LIN {X 0,Y 516.696,Z 376.127,A -85,B 0,C 180,E1 -4916.105,E2 -4916.105} C_VEL
LIN {X 0,Y 516.601,Z 376.349,A -85,B 0,C 180,E1 -4917.032,E2 -4917.032} C_VEL
LIN {X 0,Y 516.544,Z 379.132,A -85,B 0,C 180,E1 -4919.774,E2 -4919.774} C_VEL
LIN {X 0,Y 516.549,Z 381.873,A -85,B 0,C 180,E1 -4922.445,E2 -4922.445} C_VEL
LIN {X 0,Y 516.453,Z 384.593,A -85,B 0,C 180,E1 -4925.048,E2 -4925.048} C_VEL
LIN {X 0,Y 516.411,Z 387.453,A -85,B 0,C 180,E1 -4927.735,E2 -4927.735} C_VEL
LIN {X 0,Y 516.331,Z 390.983,A -85,B 0,C 180,E1 -4930.933,E2 -4930.933} C_VEL
LIN {X 0,Y 516.302,Z 393.789,A -85,B 0,C 180,E1 -4933.39,E2 -4933.39} C_VEL
LIN {X 0,Y 516.34,Z 397.21,A -85,B 0,C 180,E1 -4936.207,E2 -4936.207} C_VEL
LIN {X 0,Y 518.472,Z 408.127,A -85,B 0,C 180,E1 -4936.552,E2 -4936.552} C_VEL
LIN {X 0,Y 518.227,Z 421.717,A -85,B 0,C 180,E1 -4937.07,E2 -4937.07} C_VEL
LIN {X 0,Y 518.019,Z 432.766,A -85,B 0,C 180,E1 -4937.643,E2 -4937.643} C_VEL
LIN {X 0,Y 517.71,Z 443.454,A -85,B 0,C 180,E1 -4938.35,E2 -4938.35} C_VEL
LIN {X 0,Y 517.416,Z 454.111,A -85,B 0,C 180,E1 -4939.236,E2 -4939.236} C_VEL
LIN {X 0,Y 517.106,Z 463.696,A -85,B 0,C 180,E1 -4940.219,E2 -4940.219} C_VEL
LIN {X 0,Y 516.91,Z 471.538,A -85,B 0,C 180,E1 -4941.202,E2 -4941.202} C_VEL
LIN {X 0,Y 516.639,Z 479.209,A -85,B 0,C 180,E1 -4942.378,E2 -4942.378} C_VEL
LIN {X 0,Y 516.493,Z 486.233,A -85,B 0,C 180,E1 -4943.751,E2 -4943.751} C_VEL
LIN {X 0,Y 516.319,Z 490.918,A -85,B 0,C 180,E1 -4944.924,E2 -4944.924} C_VEL
LIN {X 0,Y 516.373,Z 494.495,A -85,B 0,C 180,E1 -4946.098,E2 -4946.098} C_VEL
LIN {X 0,Y 516.313,Z 496.349,A -85,B 0,C 180,E1 -4946.879,E2 -4946.879} C_VEL
LIN {X 0,Y 516.261,Z 497.749,A -85,B 0,C 180,E1 -4947.659,E2 -4947.659} C_VEL
LIN {X 0,Y 516.164,Z 499.358,A -85,B 0,C 180,E1 -4949.22,E2 -4949.22} C_VEL
LIN {X 0,Y 516.161,Z 499.594,A -85,B 0,C 180,E1 -4950,E2 -4950} C_VEL
LIN {X 0,Y 516.164,Z 499.412,A -85,B 0,C 180,E1 -4950.78,E2 -4950.78} C_VEL
LIN {X 0,Y 516.262,Z 497.873,A -85,B 0,C 180,E1 -4952.341,E2 -4952.341} C_VEL
LIN {X 0,Y 516.313,Z 496.527,A -85,B 0,C 180,E1 -4953.121,E2 -4953.121} C_VEL
LIN {X 0,Y 516.363,Z 493.686,A -85,B 0,C 180,E1 -4954.293,E2 -4954.293} C_VEL
LIN {X 0,Y 516.404,Z 489.833,A -85,B 0,C 180,E1 -4955.467,E2 -4955.467} C_VEL
LIN {X 0,Y 516.498,Z 483.973,A -85,B 0,C 180,E1 -4956.823,E2 -4956.823} C_VEL
LIN {X 0,Y 516.73,Z 477.373,A -85,B 0,C 180,E1 -4958.014,E2 -4958.014} C_VEL
LIN {X 0,Y 516.885,Z 469.272,A -85,B 0,C 180,E1 -4959.193,E2 -4959.193} C_VEL
LIN {X 0,Y 517.196,Z 460.967,A -85,B 0,C 180,E1 -4960.175,E2 -4960.175} C_VEL
LIN {X 0,Y 517.521,Z 450.709,A -85,B 0,C 180,E1 -4961.158,E2 -4961.158} C_VEL
LIN {X 0,Y 517.828,Z 440.101,A -85,B 0,C 180,E1 -4961.976,E2 -4961.976} C_VEL
LIN {X 0,Y 518.061,Z 429.415,A -85,B 0,C 180,E1 -4962.636,E2 -4962.636} C_VEL
LIN {X 0,Y 518.325,Z 416.909,A -85,B 0,C 180,E1 -4963.227,E2 -4963.227} C_VEL
LIN {X 0,Y 518.289,Z 407.077,A -85,B 0,C 180,E1 -4963.578,E2 -4963.578} C_VEL
LIN {X 0,Y 516.314,Z 396.997,A -85,B 0,C 180,E1 -4963.906,E2 -4963.906} C_VEL
LIN {X 0,Y 516.316,Z 393.895,A -85,B 0,C 180,E1 -4966.61,E2 -4966.61} C_VEL
LIN {X 0,Y 516.331,Z 391.104,A -85,B 0,C 180,E1 -4969.067,E2 -4969.067} C_VEL
LIN {X 0,Y 516.358,Z 388.318,A -85,B 0,C 180,E1 -4971.561,E2 -4971.561} C_VEL
LIN {X 0,Y 516.434,Z 385.383,A -85,B 0,C 180,E1 -4974.247,E2 -4974.247} C_VEL
LIN {X 0,Y 516.479,Z 382.856,A -85,B 0,C 180,E1 -4976.683,E2 -4976.683} C_VEL
LIN {X 0,Y 516.537,Z 380.02,A -85,B 0,C 180,E1 -4979.45,E2 -4979.45} C_VEL
LIN {X 0,Y 516.572,Z 377.382,A -85,B 0,C 180,E1 -4982.046,E2 -4982.046} C_VEL
LIN {X 0,Y 516.602,Z 376.437,A -85,B 0,C 180,E1 -4982.968,E2 -4982.968} C_VEL
LIN {X 0,Y 516.803,Z 376.111,A -85,B 0,C 180,E1 -4985.319,E2 -4985.319} C_VEL
LIN {X 0,Y 516.884,Z 376.098,A -85,B 0,C 180,E1 -4987.943,E2 -4987.943} C_VEL
LIN {X 0,Y 516.888,Z 376.1,A -85,B 0,C 180,E1 -4990.742,E2 -4990.742} C_VEL
LIN {X 0,Y 516.888,Z 376.098,A -85,B 0,C 180,E1 -4992.831,E2 -4992.831} C_VEL
LIN {X 0,Y 516.899,Z 376.097,A -85,B 0,C 180,E1 -4995.007,E2 -4995.007} C_VEL
LIN {X 0,Y 516.918,Z 376.095,A -85,B 0,C 180,E1 -4998.399,E2 -4998.399} C_VEL
LIN {X 0,Y 516.887,Z 376.098,A -85,B 0,C 180,E1 -5001.284,E2 -5001.284} C_VEL
LIN {X 0,Y 516.892,Z 376.103,A -85,B 0,C 180,E1 -5004.221,E2 -5004.221} C_VEL
LIN {X 0,Y 516.9,Z 376.097,A -85,B 0,C 180,E1 -5007.053,E2 -5007.053} C_VEL
LIN {X 0,Y 516.897,Z 376.099,A -85,B 0,C 180,E1 -5009.796,E2 -5009.796} C_VEL
LIN {X 0,Y 516.931,Z 376.096,A -85,B 0,C 180,E1 -5012.467,E2 -5012.467} C_VEL
LIN {X 0,Y 516.88,Z 376.098,A -85,B 0,C 180,E1 -5015.07,E2 -5015.07} C_VEL
LIN {X 0,Y 516.874,Z 376.101,A -85,B 0,C 180,E1 -5017.622,E2 -5017.622} C_VEL
LIN {X 0,Y 516.938,Z 376.093,A -85,B 0,C 180,E1 -5020.13,E2 -5020.13} C_VEL
LIN {X 0,Y 516.912,Z 376.097,A -85,B 0,C 180,E1 -5022.595,E2 -5022.595} C_VEL
LIN {X 0,Y 516.948,Z 376.093,A -85,B 0,C 180,E1 -5025.03,E2 -5025.03} C_VEL
LIN {X 0,Y 516.971,Z 376.091,A -85,B 0,C 180,E1 -5028.234,E2 -5028.234} C_VEL
LIN {X 0,Y 516.962,Z 376.091,A -85,B 0,C 180,E1 -5031.399,E2 -5031.399} C_VEL
LIN {X 0,Y 517.015,Z 376.083,A -85,B 0,C 180,E1 -5033.757,E2 -5033.757} C_VEL
LIN {X 0,Y 517.086,Z 376.074,A -85,B 0,C 180,E1 -5037.663,E2 -5037.663} C_VEL
LIN {X 0,Y 517.099,Z 376.071,A -85,B 0,C 180,E1 -5040.779,E2 -5040.779} C_VEL
LIN {X 0,Y 517.016,Z 376.082,A -85,B 0,C 180,E1 -5043.117,E2 -5043.117} C_VEL
LIN {X 0,Y 517.015,Z 376.082,A -85,B 0,C 180,E1 -5046.243,E2 -5046.243} C_VEL
LIN {X 0,Y 516.958,Z 376.09,A -85,B 0,C 180,E1 -5049.389,E2 -5049.389} C_VEL
LIN {X 0,Y 516.99,Z 376.089,A -85,B 0,C 180,E1 -5051.824,E2 -5051.824} C_VEL
LIN {X 0,Y 516.95,Z 376.091,A -85,B 0,C 180,E1 -5055.146,E2 -5055.146} C_VEL
LIN {X 0,Y 516.922,Z 376.093,A -85,B 0,C 180,E1 -5058.222,E2 -5058.222} C_VEL
LIN {X 0,Y 516.918,Z 376.098,A -85,B 0,C 180,E1 -5060.701,E2 -5060.701} C_VEL
LIN {X 0,Y 516.896,Z 376.1,A -85,B 0,C 180,E1 -5064.073,E2 -5064.073} C_VEL
LIN {X 0,Y 516.931,Z 376.092,A -85,B 0,C 180,E1 -5066.658,E2 -5066.658} C_VEL
LIN {X 0,Y 516.916,Z 376.096,A -85,B 0,C 180,E1 -5069.524,E2 -5069.524} C_VEL
LIN {X 0,Y 516.9,Z 376.099,A -85,B 0,C 180,E1 -5072.543,E2 -5072.543} C_VEL
LIN {X 0,Y 516.871,Z 376.101,A -85,B 0,C 180,E1 -5075.33,E2 -5075.33} C_VEL
LIN {X 0,Y 516.885,Z 376.1,A -85,B 0,C 180,E1 -5077.943,E2 -5077.943} C_VEL
LIN {X 0,Y 516.887,Z 376.099,A -85,B 0,C 180,E1 -5080.741,E2 -5080.741} C_VEL
LIN {X 0,Y 516.888,Z 376.103,A -85,B 0,C 180,E1 -5082.831,E2 -5082.831} C_VEL
LIN {X 0,Y 516.927,Z 376.095,A -85,B 0,C 180,E1 -5085.01,E2 -5085.01} C_VEL
LIN {X 0,Y 516.92,Z 376.097,A -85,B 0,C 180,E1 -5088.398,E2 -5088.398} C_VEL
LIN {X 0,Y 516.92,Z 376.225,A -85,B 0,C 180,E1 -5091.437,E2 -5091.437} C_VEL
LIN {X 0,Y 518.012,Z 382.521,A -85,B 0,C 180,E1 -5093.83,E2 -5093.83} C_VEL
LIN {X 0,Y 518.066,Z 388.18,A -85,B 0,C 180,E1 -5095.845,E2 -5095.845} C_VEL
LIN {X 0,Y 517.809,Z 396.871,A -85,B 0,C 180,E1 -5098.768,E2 -5098.768} C_VEL
LIN {X 0,Y 517.58,Z 406.618,A -85,B 0,C 180,E1 -5101.959,E2 -5101.959} C_VEL
LIN {X 0,Y 517.332,Z 414.957,A -85,B 0,C 180,E1 -5104.663,E2 -5104.663} C_VEL
LIN {X 0,Y 517.117,Z 424.224,A -85,B 0,C 180,E1 -5107.633,E2 -5107.633} C_VEL
LIN {X 0,Y 516.907,Z 433.491,A -85,B 0,C 180,E1 -5110.542,E2 -5110.542} C_VEL
LIN {X 0,Y 516.714,Z 442.759,A -85,B 0,C 180,E1 -5113.403,E2 -5113.403} C_VEL
LIN {X 0,Y 516.609,Z 451.72,A -85,B 0,C 180,E1 -5116.095,E2 -5116.095} C_VEL
LIN {X 0,Y 518.494,Z 463.261,A -85,B 0,C 180,E1 -5116.403,E2 -5116.403} C_VEL
LIN {X 0,Y 518.294,Z 475.766,A -85,B 0,C 180,E1 -5116.822,E2 -5116.822} C_VEL
LIN {X 0,Y 518.024,Z 487.407,A -85,B 0,C 180,E1 -5117.363,E2 -5117.363} C_VEL
LIN {X 0,Y 517.721,Z 499.455,A -85,B 0,C 180,E1 -5118.102,E2 -5118.102} C_VEL
LIN {X 0,Y 517.44,Z 510.26,A -85,B 0,C 180,E1 -5118.939,E2 -5118.939} C_VEL
LIN {X 0,Y 517.083,Z 519.537,A -85,B 0,C 180,E1 -5119.823,E2 -5119.823} C_VEL
LIN {X 0,Y 516.868,Z 527.99,A -85,B 0,C 180,E1 -5120.806,E2 -5120.806} C_VEL
LIN {X 0,Y 516.641,Z 536.236,A -85,B 0,C 180,E1 -5121.985,E2 -5121.985} C_VEL
LIN {X 0,Y 516.48,Z 543.077,A -85,B 0,C 180,E1 -5123.201,E2 -5123.201} C_VEL
LIN {X 0,Y 516.405,Z 548.949,A -85,B 0,C 180,E1 -5124.533,E2 -5124.533} C_VEL
LIN {X 0,Y 516.343,Z 552.895,A -85,B 0,C 180,E1 -5125.707,E2 -5125.707} C_VEL
LIN {X 0,Y 516.282,Z 555.807,A -85,B 0,C 180,E1 -5126.879,E2 -5126.879} C_VEL
LIN {X 0,Y 516.261,Z 557.196,A -85,B 0,C 180,E1 -5127.659,E2 -5127.659} C_VEL
LIN {X 0,Y 516.16,Z 558.785,A -85,B 0,C 180,E1 -5129.22,E2 -5129.22} C_VEL
LIN {X 0,Y 516.154,Z 559,A -85,B 0,C 180,E1 -5130,E2 -5130} C_VEL
LIN {X 0,Y 516.192,Z 558.185,A -85,B 0,C 180,E1 -5131.56,E2 -5131.56} C_VEL
LIN {X 0,Y 516.261,Z 557.198,A -85,B 0,C 180,E1 -5132.341,E2 -5132.341} C_VEL
LIN {X 0,Y 516.282,Z 555.81,A -85,B 0,C 180,E1 -5133.121,E2 -5133.121} C_VEL
LIN {X 0,Y 516.343,Z 552.896,A -85,B 0,C 180,E1 -5134.293,E2 -5134.293} C_VEL
LIN {X 0,Y 516.405,Z 548.949,A -85,B 0,C 180,E1 -5135.467,E2 -5135.467} C_VEL
LIN {X 0,Y 516.486,Z 543.034,A -85,B 0,C 180,E1 -5136.807,E2 -5136.807} C_VEL
LIN {X 0,Y 516.641,Z 536.237,A -85,B 0,C 180,E1 -5138.015,E2 -5138.015} C_VEL
LIN {X 0,Y 516.868,Z 527.991,A -85,B 0,C 180,E1 -5139.193,E2 -5139.193} C_VEL
LIN {X 0,Y 517.083,Z 519.539,A -85,B 0,C 180,E1 -5140.177,E2 -5140.177} C_VEL
LIN {X 0,Y 517.477,Z 509.096,A -85,B 0,C 180,E1 -5141.159,E2 -5141.159} C_VEL
LIN {X 0,Y 517.73,Z 497.546,A -85,B 0,C 180,E1 -5142.032,E2 -5142.032} C_VEL
LIN {X 0,Y 518.08,Z 485.488,A -85,B 0,C 180,E1 -5142.735,E2 -5142.735} C_VEL
LIN {X 0,Y 518.362,Z 473.168,A -85,B 0,C 180,E1 -5143.276,E2 -5143.276} C_VEL
LIN {X 0,Y 518.314,Z 461.889,A -85,B 0,C 180,E1 -5143.639,E2 -5143.639} C_VEL
LIN {X 0,Y 516.593,Z 451.53,A -85,B 0,C 180,E1 -5143.924,E2 -5143.924} C_VEL
LIN {X 0,Y 516.714,Z 442.759,A -85,B 0,C 180,E1 -5146.596,E2 -5146.596} C_VEL
LIN {X 0,Y 516.906,Z 433.492,A -85,B 0,C 180,E1 -5149.458,E2 -5149.458} C_VEL
LIN {X 0,Y 517.102,Z 423.96,A -85,B 0,C 180,E1 -5152.452,E2 -5152.452} C_VEL
LIN {X 0,Y 517.334,Z 414.957,A -85,B 0,C 180,E1 -5155.336,E2 -5155.336} C_VEL
LIN {X 0,Y 517.607,Z 405.58,A -85,B 0,C 180,E1 -5158.374,E2 -5158.374} C_VEL
LIN {X 0,Y 517.859,Z 395.917,A -85,B 0,C 180,E1 -5161.551,E2 -5161.551} C_VEL
LIN {X 0,Y 518.059,Z 388.196,A -85,B 0,C 180,E1 -5164.154,E2 -5164.154} C_VEL
LIN {X 0,Y 518.018,Z 382.482,A -85,B 0,C 180,E1 -5166.169,E2 -5166.169} C_VEL
LIN {X 0,Y 516.898,Z 376.102,A -85,B 0,C 180,E1 -5168.615,E2 -5168.615} C_VEL
LIN {X 0,Y 516.917,Z 376.1,A -85,B 0,C 180,E1 -5171.775,E2 -5171.775} C_VEL
LIN {X 0,Y 516.926,Z 376.099,A -85,B 0,C 180,E1 -5175.01,E2 -5175.01} C_VEL
LIN {X 0,Y 516.918,Z 376.094,A -85,B 0,C 180,E1 -5178.399,E2 -5178.399} C_VEL
LIN {X 0,Y 516.886,Z 376.098,A -85,B 0,C 180,E1 -5181.284,E2 -5181.284} C_VEL
LIN {X 0,Y 516.89,Z 376.102,A -85,B 0,C 180,E1 -5184.221,E2 -5184.221} C_VEL
LIN {X 0,Y 516.898,Z 376.099,A -85,B 0,C 180,E1 -5187.053,E2 -5187.053} C_VEL
LIN {X 0,Y 516.896,Z 376.096,A -85,B 0,C 180,E1 -5189.796,E2 -5189.796} C_VEL
LIN {X 0,Y 516.932,Z 376.096,A -85,B 0,C 180,E1 -5192.467,E2 -5192.467} C_VEL
LIN {X 0,Y 516.879,Z 376.099,A -85,B 0,C 180,E1 -5195.07,E2 -5195.07} C_VEL
LIN {X 0,Y 516.872,Z 376.103,A -85,B 0,C 180,E1 -5197.622,E2 -5197.622} C_VEL
LIN {X 0,Y 516.936,Z 376.092,A -85,B 0,C 180,E1 -5200.13,E2 -5200.13} C_VEL
LIN {X 0,Y 516.933,Z 376.095,A -85,B 0,C 180,E1 -5202.596,E2 -5202.596} C_VEL
LIN {X 0,Y 516.947,Z 376.09,A -85,B 0,C 180,E1 -5205.03,E2 -5205.03} C_VEL
LIN {X 0,Y 517.009,Z 376.086,A -85,B 0,C 180,E1 -5208.235,E2 -5208.235} C_VEL
LIN {X 0,Y 516.974,Z 376.09,A -85,B 0,C 180,E1 -5211.4,E2 -5211.4} C_VEL
LIN {X 0,Y 517.014,Z 376.082,A -85,B 0,C 180,E1 -5213.757,E2 -5213.757} C_VEL
LIN {X 0,Y 517.088,Z 376.072,A -85,B 0,C 180,E1 -5217.663,E2 -5217.663} C_VEL
LIN {X 0,Y 517.097,Z 376.072,A -85,B 0,C 180,E1 -5220.779,E2 -5220.779} C_VEL
LIN {X 0,Y 517.015,Z 376.085,A -85,B 0,C 180,E1 -5223.117,E2 -5223.117} C_VEL
LIN {X 0,Y 517.014,Z 376.083,A -85,B 0,C 180,E1 -5226.243,E2 -5226.243} C_VEL
LIN {X 0,Y 516.947,Z 376.089,A -85,B 0,C 180,E1 -5229.389,E2 -5229.389} C_VEL
LIN {X 0,Y 516.957,Z 376.092,A -85,B 0,C 180,E1 -5231.807,E2 -5231.807} C_VEL
LIN {X 0,Y 516.949,Z 376.093,A -85,B 0,C 180,E1 -5235.147,E2 -5235.147} C_VEL
LIN {X 0,Y 516.921,Z 376.095,A -85,B 0,C 180,E1 -5238.222,E2 -5238.222} C_VEL
LIN {X 0,Y 516.917,Z 376.096,A -85,B 0,C 180,E1 -5240.701,E2 -5240.701} C_VEL
LIN {X 0,Y 516.895,Z 376.1,A -85,B 0,C 180,E1 -5244.073,E2 -5244.073} C_VEL
LIN {X 0,Y 516.93,Z 376.093,A -85,B 0,C 180,E1 -5246.658,E2 -5246.658} C_VEL
LIN {X 0,Y 516.915,Z 376.096,A -85,B 0,C 180,E1 -5249.524,E2 -5249.524} C_VEL
LIN {X 0,Y 516.899,Z 376.099,A -85,B 0,C 180,E1 -5252.543,E2 -5252.543} C_VEL
LIN {X 0,Y 516.87,Z 376.1,A -85,B 0,C 180,E1 -5255.33,E2 -5255.33} C_VEL
LIN {X 0,Y 516.885,Z 376.1,A -85,B 0,C 180,E1 -5257.943,E2 -5257.943} C_VEL
LIN {X 0,Y 516.888,Z 376.1,A -85,B 0,C 180,E1 -5260.742,E2 -5260.742} C_VEL
LIN {X 0,Y 516.886,Z 376.101,A -85,B 0,C 180,E1 -5262.831,E2 -5262.831} C_VEL
LIN {X 0,Y 516.886,Z 376.102,A -85,B 0,C 180,E1 -5266.097,E2 -5266.097} C_VEL
LIN {X 0,Y 516.919,Z 376.093,A -85,B 0,C 180,E1 -5268.398,E2 -5268.398} C_VEL
LIN {X 0,Y 516.884,Z 376.097,A -85,B 0,C 180,E1 -5270.3,E2 -5270.3} C_VEL
LIN {X 0,Y 516.212,Z 376.184,A -85,B 0,C 180,E1 -5270.95,E2 -5270.95} C_VEL
LIN {X 0,Y 513.358,Z 376.538,A -85,B 0,C 180,E1 -5272.006,E2 -5272.006} C_VEL
LIN {X 0,Y 510.936,Z 376.842,A -85,B 0,C 180,E1 -5272.856,E2 -5272.856} C_VEL
LIN {X 0,Y 509.877,Z 376.973,A -85,B 0,C 180,E1 -5273.512,E2 -5273.512} C_VEL
LIN {X 0,Y 509.781,Z 376.983,A -85,B 0,C 180,E1 -5273.735,E2 -5273.735} C_VEL
LIN {X 0,Y 509.584,Z 377.013,A -85,B 0,C 180,E1 -5276.519,E2 -5276.519} C_VEL
LIN {X 0,Y 509.535,Z 377.482,A -85,B 0,C 180,E1 -5277.457,E2 -5277.457} C_VEL
LIN {X 0,Y 509.477,Z 380.405,A -85,B 0,C 180,E1 -5280.35,E2 -5280.35} C_VEL
LIN {X 0,Y 509.428,Z 383.029,A -85,B 0,C 180,E1 -5282.918,E2 -5282.918} C_VEL
LIN {X 0,Y 509.385,Z 385.793,A -85,B 0,C 180,E1 -5285.59,E2 -5285.59} C_VEL
LIN {X 0,Y 509.309,Z 388.47,A -85,B 0,C 180,E1 -5288.125,E2 -5288.125} C_VEL
LIN {X 0,Y 509.257,Z 391.242,A -85,B 0,C 180,E1 -5290.658,E2 -5290.658} C_VEL
LIN {X 0,Y 509.242,Z 394.076,A -85,B 0,C 180,E1 -5293.153,E2 -5293.153} C_VEL
LIN {X 0,Y 509.28,Z 397.682,A -85,B 0,C 180,E1 -5296.012,E2 -5296.012} C_VEL
LIN {X 0,Y 511.461,Z 408.207,A -85,B 0,C 180,E1 -5296.352,E2 -5296.352} C_VEL
LIN {X 0,Y 511.394,Z 421.035,A -85,B 0,C 180,E1 -5296.843,E2 -5296.843} C_VEL
LIN {X 0,Y 511.133,Z 432.226,A -85,B 0,C 180,E1 -5297.418,E2 -5297.418} C_VEL
LIN {X 0,Y 510.776,Z 443.894,A -85,B 0,C 180,E1 -5298.19,E2 -5298.19} C_VEL
LIN {X 0,Y 510.46,Z 454.549,A -85,B 0,C 180,E1 -5299.088,E2 -5299.088} C_VEL
LIN {X 0,Y 510.137,Z 464.132,A -85,B 0,C 180,E1 -5300.084,E2 -5300.084} C_VEL
LIN {X 0,Y 509.914,Z 471.974,A -85,B 0,C 180,E1 -5301.08,E2 -5301.08} C_VEL
LIN {X 0,Y 509.611,Z 479.644,A -85,B 0,C 180,E1 -5302.273,E2 -5302.273} C_VEL
LIN {X 0,Y 509.445,Z 486.667,A -85,B 0,C 180,E1 -5303.664,E2 -5303.664} C_VEL
LIN {X 0,Y 509.256,Z 491.352,A -85,B 0,C 180,E1 -5304.854,E2 -5304.854} C_VEL
LIN {X 0,Y 509.304,Z 494.928,A -85,B 0,C 180,E1 -5306.044,E2 -5306.044} C_VEL
LIN {X 0,Y 509.259,Z 496.78,A -85,B 0,C 180,E1 -5306.836,E2 -5306.836} C_VEL
LIN {X 0,Y 509.191,Z 498.18,A -85,B 0,C 180,E1 -5307.627,E2 -5307.627} C_VEL
LIN {X 0,Y 509.079,Z 499.79,A -85,B 0,C 180,E1 -5309.209,E2 -5309.209} C_VEL
LIN {X 0,Y 509.075,Z 500.026,A -85,B 0,C 180,E1 -5310,E2 -5310} C_VEL
LIN {X 0,Y 509.078,Z 499.843,A -85,B 0,C 180,E1 -5310.791,E2 -5310.791} C_VEL
LIN {X 0,Y 509.192,Z 498.303,A -85,B 0,C 180,E1 -5312.373,E2 -5312.373} C_VEL
LIN {X 0,Y 509.26,Z 496.956,A -85,B 0,C 180,E1 -5313.165,E2 -5313.165} C_VEL
LIN {X 0,Y 509.291,Z 494.116,A -85,B 0,C 180,E1 -5314.353,E2 -5314.353} C_VEL
LIN {X 0,Y 509.346,Z 490.262,A -85,B 0,C 180,E1 -5315.543,E2 -5315.543} C_VEL
LIN {X 0,Y 509.467,Z 484.594,A -85,B 0,C 180,E1 -5316.879,E2 -5316.879} C_VEL
LIN {X 0,Y 509.702,Z 477.802,A -85,B 0,C 180,E1 -5318.125,E2 -5318.125} C_VEL
LIN {X 0,Y 509.894,Z 469.699,A -85,B 0,C 180,E1 -5319.32,E2 -5319.32} C_VEL
LIN {X 0,Y 510.24,Z 461.391,A -85,B 0,C 180,E1 -5320.315,E2 -5320.315} C_VEL
LIN {X 0,Y 510.578,Z 451.132,A -85,B 0,C 180,E1 -5321.312,E2 -5321.312} C_VEL
LIN {X 0,Y 510.933,Z 439.931,A -85,B 0,C 180,E1 -5322.182,E2 -5322.182} C_VEL
LIN {X 0,Y 511.212,Z 428.023,A -85,B 0,C 180,E1 -5322.909,E2 -5322.909} C_VEL
LIN {X 0,Y 511.496,Z 416.025,A -85,B 0,C 180,E1 -5323.458,E2 -5323.458} C_VEL
LIN {X 0,Y 511.373,Z 407.878,A -85,B 0,C 180,E1 -5323.752,E2 -5323.752} C_VEL
LIN {X 0,Y 509.272,Z 397.377,A -85,B 0,C 180,E1 -5324.103,E2 -5324.103} C_VEL
LIN {X 0,Y 509.308,Z 393.254,A -85,B 0,C 180,E1 -5327.673,E2 -5327.673} C_VEL
LIN {X 0,Y 509.265,Z 389.476,A -85,B 0,C 180,E1 -5331.027,E2 -5331.027} C_VEL
LIN {X 0,Y 509.334,Z 386.717,A -85,B 0,C 180,E1 -5333.588,E2 -5333.588} C_VEL
LIN {X 0,Y 509.412,Z 383.937,A -85,B 0,C 180,E1 -5336.264,E2 -5336.264} C_VEL
LIN {X 0,Y 509.475,Z 381.285,A -85,B 0,C 180,E1 -5338.869,E2 -5338.869} C_VEL
LIN {X 0,Y 509.515,Z 378.508,A -85,B 0,C 180,E1 -5341.612,E2 -5341.612} C_VEL
LIN {X 0,Y 509.538,Z 377.403,A -85,B 0,C 180,E1 -5342.715,E2 -5342.715} C_VEL
LIN {X 0,Y 509.653,Z 377.004,A -85,B 0,C 180,E1 -5344.168,E2 -5344.168} C_VEL
LIN {X 0,Y 509.799,Z 376.985,A -85,B 0,C 180,E1 -5346.91,E2 -5346.91} C_VEL
LIN {X 0,Y 509.838,Z 376.975,A -85,B 0,C 180,E1 -5349.471,E2 -5349.471} C_VEL
LIN {X 0,Y 509.839,Z 376.979,A -85,B 0,C 180,E1 -5352.49,E2 -5352.49} C_VEL
LIN {X 0,Y 509.843,Z 376.978,A -85,B 0,C 180,E1 -5355.33,E2 -5355.33} C_VEL
LIN {X 0,Y 509.86,Z 376.975,A -85,B 0,C 180,E1 -5358.575,E2 -5358.575} C_VEL
LIN {X 0,Y 509.856,Z 376.973,A -85,B 0,C 180,E1 -5361.786,E2 -5361.786} C_VEL
LIN {X 0,Y 509.847,Z 376.975,A -85,B 0,C 180,E1 -5364.623,E2 -5364.623} C_VEL
LIN {X 0,Y 509.866,Z 376.975,A -85,B 0,C 180,E1 -5367.481,E2 -5367.481} C_VEL
LIN {X 0,Y 509.863,Z 376.974,A -85,B 0,C 180,E1 -5370.274,E2 -5370.274} C_VEL
LIN {X 0,Y 509.889,Z 376.972,A -85,B 0,C 180,E1 -5372.944,E2 -5372.944} C_VEL
LIN {X 0,Y 509.856,Z 376.973,A -85,B 0,C 180,E1 -5375.573,E2 -5375.573} C_VEL
LIN {X 0,Y 509.827,Z 376.98,A -85,B 0,C 180,E1 -5378.149,E2 -5378.149} C_VEL
LIN {X 0,Y 509.869,Z 376.973,A -85,B 0,C 180,E1 -5380.682,E2 -5380.682} C_VEL
LIN {X 0,Y 509.879,Z 376.974,A -85,B 0,C 180,E1 -5383.174,E2 -5383.174} C_VEL
LIN {X 0,Y 509.87,Z 376.972,A -85,B 0,C 180,E1 -5385.634,E2 -5385.634} C_VEL
LIN {X 0,Y 509.918,Z 376.965,A -85,B 0,C 180,E1 -5388.875,E2 -5388.875} C_VEL
LIN {X 0,Y 509.927,Z 376.966,A -85,B 0,C 180,E1 -5392.078,E2 -5392.078} C_VEL
LIN {X 0,Y 509.987,Z 376.959,A -85,B 0,C 180,E1 -5394.464,E2 -5394.464} C_VEL
LIN {X 0,Y 510.058,Z 376.949,A -85,B 0,C 180,E1 -5397.631,E2 -5397.631} C_VEL
LIN {X 0,Y 510.069,Z 376.947,A -85,B 0,C 180,E1 -5400.789,E2 -5400.789} C_VEL
LIN {X 0,Y 509.958,Z 376.961,A -85,B 0,C 180,E1 -5403.16,E2 -5403.16} C_VEL
LIN {X 0,Y 509.983,Z 376.958,A -85,B 0,C 180,E1 -5406.33,E2 -5406.33} C_VEL
LIN {X 0,Y 509.921,Z 376.969,A -85,B 0,C 180,E1 -5408.72,E2 -5408.72} C_VEL
LIN {X 0,Y 509.957,Z 376.966,A -85,B 0,C 180,E1 -5411.93,E2 -5411.93} C_VEL
LIN {X 0,Y 509.899,Z 376.97,A -85,B 0,C 180,E1 -5415.242,E2 -5415.242} C_VEL
LIN {X 0,Y 509.867,Z 376.973,A -85,B 0,C 180,E1 -5418.484,E2 -5418.484} C_VEL
LIN {X 0,Y 509.856,Z 376.977,A -85,B 0,C 180,E1 -5421.001,E2 -5421.001} C_VEL
LIN {X 0,Y 509.827,Z 376.979,A -85,B 0,C 180,E1 -5423.564,E2 -5423.564} C_VEL
LIN {X 0,Y 509.917,Z 376.966,A -85,B 0,C 180,E1 -5426.378,E2 -5426.378} C_VEL
LIN {X 0,Y 509.882,Z 376.971,A -85,B 0,C 180,E1 -5428.844,E2 -5428.844} C_VEL
LIN {X 0,Y 509.824,Z 376.978,A -85,B 0,C 180,E1 -5431.59,E2 -5431.59} C_VEL
LIN {X 0,Y 509.852,Z 376.977,A -85,B 0,C 180,E1 -5434.414,E2 -5434.414} C_VEL
LIN {X 0,Y 509.821,Z 376.981,A -85,B 0,C 180,E1 -5437.341,E2 -5437.341} C_VEL
LIN {X 0,Y 509.842,Z 376.975,A -85,B 0,C 180,E1 -5440.382,E2 -5440.382} C_VEL
LIN {X 0,Y 509.828,Z 376.982,A -85,B 0,C 180,E1 -5443.062,E2 -5443.062} C_VEL
LIN {X 0,Y 509.835,Z 376.978,A -85,B 0,C 180,E1 -5445.792,E2 -5445.792} C_VEL
LIN {X 0,Y 509.861,Z 376.975,A -85,B 0,C 180,E1 -5448.575,E2 -5448.575} C_VEL
LIN {X 0,Y 509.855,Z 377.034,A -85,B 0,C 180,E1 -5451.157,E2 -5451.157} C_VEL
LIN {X 0,Y 511.036,Z 383.679,A -85,B 0,C 180,E1 -5453.746,E2 -5453.746} C_VEL
LIN {X 0,Y 511.083,Z 389.074,A -85,B 0,C 180,E1 -5455.681,E2 -5455.681} C_VEL
LIN {X 0,Y 510.85,Z 397.384,A -85,B 0,C 180,E1 -5458.536,E2 -5458.536} C_VEL
LIN {X 0,Y 510.567,Z 407.086,A -85,B 0,C 180,E1 -5461.759,E2 -5461.759} C_VEL
LIN {X 0,Y 510.31,Z 416.281,A -85,B 0,C 180,E1 -5464.727,E2 -5464.727} C_VEL
LIN {X 0,Y 510.081,Z 425.671,A -85,B 0,C 180,E1 -5467.774,E2 -5467.774} C_VEL
LIN {X 0,Y 509.859,Z 434.815,A -85,B 0,C 180,E1 -5470.681,E2 -5470.681} C_VEL
LIN {X 0,Y 509.65,Z 445.407,A -85,B 0,C 180,E1 -5473.99,E2 -5473.99} C_VEL
LIN {X 0,Y 509.563,Z 451.72,A -85,B 0,C 180,E1 -5475.899,E2 -5475.899} C_VEL
LIN {X 0,Y 511.588,Z 464.176,A -85,B 0,C 180,E1 -5476.241,E2 -5476.241} C_VEL
LIN {X 0,Y 511.355,Z 476.979,A -85,B 0,C 180,E1 -5476.69,E2 -5476.69} C_VEL
LIN {X 0,Y 511.034,Z 489.171,A -85,B 0,C 180,E1 -5477.288,E2 -5477.288} C_VEL
LIN {X 0,Y 510.751,Z 499.859,A -85,B 0,C 180,E1 -5477.965,E2 -5477.965} C_VEL
LIN {X 0,Y 510.474,Z 510.261,A -85,B 0,C 180,E1 -5478.786,E2 -5478.786} C_VEL
LIN {X 0,Y 510.072,Z 519.537,A -85,B 0,C 180,E1 -5479.681,E2 -5479.681} C_VEL
LIN {X 0,Y 509.846,Z 527.99,A -85,B 0,C 180,E1 -5480.679,E2 -5480.679} C_VEL
LIN {X 0,Y 509.585,Z 536.235,A -85,B 0,C 180,E1 -5481.873,E2 -5481.873} C_VEL
LIN {X 0,Y 509.419,Z 542.876,A -85,B 0,C 180,E1 -5483.067,E2 -5483.067} C_VEL
LIN {X 0,Y 509.344,Z 548.949,A -85,B 0,C 180,E1 -5484.457,E2 -5484.457} C_VEL
LIN {X 0,Y 509.234,Z 552.894,A -85,B 0,C 180,E1 -5485.647,E2 -5485.647} C_VEL
LIN {X 0,Y 509.2,Z 555.807,A -85,B 0,C 180,E1 -5486.835,E2 -5486.835} C_VEL
LIN {X 0,Y 509.161,Z 557.196,A -85,B 0,C 180,E1 -5487.627,E2 -5487.627} C_VEL
LIN {X 0,Y 509.073,Z 558.786,A -85,B 0,C 180,E1 -5489.209,E2 -5489.209} C_VEL
LIN {X 0,Y 509.065,Z 559,A -85,B 0,C 180,E1 -5490,E2 -5490} C_VEL
LIN {X 0,Y 509.113,Z 558.185,A -85,B 0,C 180,E1 -5491.582,E2 -5491.582} C_VEL
LIN {X 0,Y 509.161,Z 557.198,A -85,B 0,C 180,E1 -5492.373,E2 -5492.373} C_VEL
LIN {X 0,Y 509.2,Z 555.81,A -85,B 0,C 180,E1 -5493.165,E2 -5493.165} C_VEL
LIN {X 0,Y 509.233,Z 552.896,A -85,B 0,C 180,E1 -5494.353,E2 -5494.353} C_VEL
LIN {X 0,Y 509.344,Z 548.949,A -85,B 0,C 180,E1 -5495.543,E2 -5495.543} C_VEL
LIN {X 0,Y 509.41,Z 543.282,A -85,B 0,C 180,E1 -5496.853,E2 -5496.853} C_VEL
LIN {X 0,Y 509.585,Z 536.237,A -85,B 0,C 180,E1 -5498.127,E2 -5498.127} C_VEL
LIN {X 0,Y 509.846,Z 527.991,A -85,B 0,C 180,E1 -5499.321,E2 -5499.321} C_VEL
LIN {X 0,Y 510.071,Z 519.539,A -85,B 0,C 180,E1 -5500.319,E2 -5500.319} C_VEL
LIN {X 0,Y 510.505,Z 509.095,A -85,B 0,C 180,E1 -5501.313,E2 -5501.313} C_VEL
LIN {X 0,Y 510.757,Z 498.326,A -85,B 0,C 180,E1 -5502.143,E2 -5502.143} C_VEL
LIN {X 0,Y 511.08,Z 487.407,A -85,B 0,C 180,E1 -5502.811,E2 -5502.811} C_VEL
LIN {X 0,Y 511.423,Z 475.763,A -85,B 0,C 180,E1 -5503.358,E2 -5503.358} C_VEL
LIN {X 0,Y 511.401,Z 462.803,A -85,B 0,C 180,E1 -5503.802,E2 -5503.802} C_VEL
LIN {X 0,Y 509.552,Z 451.53,A -85,B 0,C 180,E1 -5504.12,E2 -5504.12} C_VEL
LIN {X 0,Y 509.718,Z 441.435,A -85,B 0,C 180,E1 -5507.244,E2 -5507.244} C_VEL
LIN {X 0,Y 509.924,Z 432.168,A -85,B 0,C 180,E1 -5510.155,E2 -5510.155} C_VEL
LIN {X 0,Y 510.125,Z 422.901,A -85,B 0,C 180,E1 -5513.119,E2 -5513.119} C_VEL
LIN {X 0,Y 510.371,Z 413.583,A -85,B 0,C 180,E1 -5516.146,E2 -5516.146} C_VEL
LIN {X 0,Y 510.588,Z 405.374,A -85,B 0,C 180,E1 -5518.8,E2 -5518.8} C_VEL
LIN {X 0,Y 510.861,Z 397.224,A -85,B 0,C 180,E1 -5521.519,E2 -5521.519} C_VEL
LIN {X 0,Y 511.09,Z 388.84,A -85,B 0,C 180,E1 -5524.405,E2 -5524.405} C_VEL
LIN {X 0,Y 511.039,Z 383.669,A -85,B 0,C 180,E1 -5526.253,E2 -5526.253} C_VEL
LIN {X 0,Y 509.86,Z 376.978,A -85,B 0,C 180,E1 -5528.906,E2 -5528.906} C_VEL
LIN {X 0,Y 509.863,Z 376.979,A -85,B 0,C 180,E1 -5531.897,E2 -5531.897} C_VEL
LIN {X 0,Y 509.86,Z 376.981,A -85,B 0,C 180,E1 -5535.332,E2 -5535.332} C_VEL
LIN {X 0,Y 509.86,Z 376.974,A -85,B 0,C 180,E1 -5538.575,E2 -5538.575} C_VEL
LIN {X 0,Y 509.855,Z 376.975,A -85,B 0,C 180,E1 -5541.786,E2 -5541.786} C_VEL
LIN {X 0,Y 509.846,Z 376.976,A -85,B 0,C 180,E1 -5544.623,E2 -5544.623} C_VEL
LIN {X 0,Y 509.864,Z 376.975,A -85,B 0,C 180,E1 -5547.481,E2 -5547.481} C_VEL
LIN {X 0,Y 509.862,Z 376.973,A -85,B 0,C 180,E1 -5550.274,E2 -5550.274} C_VEL
LIN {X 0,Y 509.889,Z 376.971,A -85,B 0,C 180,E1 -5552.945,E2 -5552.945} C_VEL
LIN {X 0,Y 509.855,Z 376.976,A -85,B 0,C 180,E1 -5555.573,E2 -5555.573} C_VEL
LIN {X 0,Y 509.826,Z 376.979,A -85,B 0,C 180,E1 -5558.149,E2 -5558.149} C_VEL
LIN {X 0,Y 509.869,Z 376.974,A -85,B 0,C 180,E1 -5560.682,E2 -5560.682} C_VEL
LIN {X 0,Y 509.888,Z 376.97,A -85,B 0,C 180,E1 -5563.175,E2 -5563.175} C_VEL
LIN {X 0,Y 509.869,Z 376.972,A -85,B 0,C 180,E1 -5565.634,E2 -5565.634} C_VEL
LIN {X 0,Y 509.926,Z 376.965,A -85,B 0,C 180,E1 -5568.875,E2 -5568.875} C_VEL
LIN {X 0,Y 509.956,Z 376.962,A -85,B 0,C 180,E1 -5572.079,E2 -5572.079} C_VEL
LIN {X 0,Y 509.985,Z 376.96,A -85,B 0,C 180,E1 -5574.464,E2 -5574.464} C_VEL
LIN {X 0,Y 510.059,Z 376.947,A -85,B 0,C 180,E1 -5577.631,E2 -5577.631} C_VEL
LIN {X 0,Y 510.068,Z 376.947,A -85,B 0,C 180,E1 -5580.79,E2 -5580.79} C_VEL
LIN {X 0,Y 509.957,Z 376.964,A -85,B 0,C 180,E1 -5583.16,E2 -5583.16} C_VEL
LIN {X 0,Y 509.982,Z 376.96,A -85,B 0,C 180,E1 -5586.33,E2 -5586.33} C_VEL
LIN {X 0,Y 509.913,Z 376.968,A -85,B 0,C 180,E1 -5588.72,E2 -5588.72} C_VEL
LIN {X 0,Y 509.909,Z 376.972,A -85,B 0,C 180,E1 -5591.932,E2 -5591.932} C_VEL
LIN {X 0,Y 509.898,Z 376.971,A -85,B 0,C 180,E1 -5595.242,E2 -5595.242} C_VEL
LIN {X 0,Y 509.871,Z 376.972,A -85,B 0,C 180,E1 -5597.993,E2 -5597.993} C_VEL
LIN {X 0,Y 509.891,Z 376.974,A -85,B 0,C 180,E1 -5600.402,E2 -5600.402} C_VEL
LIN {X 0,Y 509.826,Z 376.978,A -85,B 0,C 180,E1 -5603.564,E2 -5603.564} C_VEL
LIN {X 0,Y 509.916,Z 376.966,A -85,B 0,C 180,E1 -5606.379,E2 -5606.379} C_VEL
LIN {X 0,Y 509.881,Z 376.973,A -85,B 0,C 180,E1 -5608.844,E2 -5608.844} C_VEL
LIN {X 0,Y 509.823,Z 376.978,A -85,B 0,C 180,E1 -5611.59,E2 -5611.59} C_VEL
LIN {X 0,Y 509.851,Z 376.976,A -85,B 0,C 180,E1 -5614.414,E2 -5614.414} C_VEL
LIN {X 0,Y 509.821,Z 376.98,A -85,B 0,C 180,E1 -5617.341,E2 -5617.341} C_VEL
LIN {X 0,Y 509.842,Z 376.976,A -85,B 0,C 180,E1 -5620.382,E2 -5620.382} C_VEL
LIN {X 0,Y 509.826,Z 376.981,A -85,B 0,C 180,E1 -5623.062,E2 -5623.062} C_VEL
LIN {X 0,Y 509.826,Z 376.98,A -85,B 0,C 180,E1 -5625.793,E2 -5625.793} C_VEL
LIN {X 0,Y 509.861,Z 376.972,A -85,B 0,C 180,E1 -5628.575,E2 -5628.575} C_VEL
LIN {X 0,Y 509.854,Z 376.975,A -85,B 0,C 180,E1 -5631.787,E2 -5631.787} C_VEL
LIN {X 0,Y 509.781,Z 376.983,A -85,B 0,C 180,E1 -5633.735,E2 -5633.735} C_VEL
LIN {X 0,Y 509.067,Z 377.098,A -85,B 0,C 180,E1 -5634.395,E2 -5634.395} C_VEL
LIN {X 0,Y 506.12,Z 377.445,A -85,B 0,C 180,E1 -5635.465,E2 -5635.465} C_VEL
LIN {X 0,Y 503.637,Z 377.753,A -85,B 0,C 180,E1 -5636.326,E2 -5636.326} C_VEL
LIN {X 0,Y 502.559,Z 377.91,A -85,B 0,C 180,E1 -5636.991,E2 -5636.991} C_VEL
LIN {X 0,Y 502.465,Z 378.038,A -85,B 0,C 180,E1 -5637.215,E2 -5637.215} C_VEL
LIN {X 0,Y 502.427,Z 380.883,A -85,B 0,C 180,E1 -5640.143,E2 -5640.143} C_VEL
LIN {X 0,Y 502.371,Z 383.283,A -85,B 0,C 180,E1 -5642.506,E2 -5642.506} C_VEL
LIN {X 0,Y 502.299,Z 386.288,A -85,B 0,C 180,E1 -5645.431,E2 -5645.431} C_VEL
LIN {X 0,Y 502.252,Z 388.748,A -85,B 0,C 180,E1 -5647.802,E2 -5647.802} C_VEL
LIN {X 0,Y 502.207,Z 391.512,A -85,B 0,C 180,E1 -5650.375,E2 -5650.375} C_VEL
LIN {X 0,Y 502.187,Z 394.385,A -85,B 0,C 180,E1 -5652.909,E2 -5652.909} C_VEL
LIN {X 0,Y 502.188,Z 397.872,A -85,B 0,C 180,E1 -5655.798,E2 -5655.798} C_VEL
LIN {X 0,Y 504.628,Z 409.413,A -85,B 0,C 180,E1 -5656.189,E2 -5656.189} C_VEL
LIN {X 0,Y 504.469,Z 422.605,A -85,B 0,C 180,E1 -5656.711,E2 -5656.711} C_VEL
LIN {X 0,Y 504.182,Z 434.63,A -85,B 0,C 180,E1 -5657.36,E2 -5657.36} C_VEL
LIN {X 0,Y 503.807,Z 445.615,A -85,B 0,C 180,E1 -5658.126,E2 -5658.126} C_VEL
LIN {X 0,Y 503.475,Z 456.048,A -85,B 0,C 180,E1 -5659.036,E2 -5659.036} C_VEL
LIN {X 0,Y 503.172,Z 464.568,A -85,B 0,C 180,E1 -5659.945,E2 -5659.945} C_VEL
LIN {X 0,Y 502.907,Z 472.41,A -85,B 0,C 180,E1 -5660.955,E2 -5660.955} C_VEL
LIN {X 0,Y 502.599,Z 480.079,A -85,B 0,C 180,E1 -5662.164,E2 -5662.164} C_VEL
LIN {X 0,Y 502.403,Z 487.102,A -85,B 0,C 180,E1 -5663.575,E2 -5663.575} C_VEL
LIN {X 0,Y 502.194,Z 491.786,A -85,B 0,C 180,E1 -5664.781,E2 -5664.781} C_VEL
LIN {X 0,Y 502.237,Z 495.361,A -85,B 0,C 180,E1 -5665.988,E2 -5665.988} C_VEL
LIN {X 0,Y 502.207,Z 497.212,A -85,B 0,C 180,E1 -5666.791,E2 -5666.791} C_VEL
LIN {X 0,Y 502.125,Z 498.612,A -85,B 0,C 180,E1 -5667.594,E2 -5667.594} C_VEL
LIN {X 0,Y 501.995,Z 500.222,A -85,B 0,C 180,E1 -5669.198,E2 -5669.198} C_VEL
LIN {X 0,Y 501.989,Z 500.457,A -85,B 0,C 180,E1 -5670,E2 -5670} C_VEL
LIN {X 0,Y 501.995,Z 500.275,A -85,B 0,C 180,E1 -5670.802,E2 -5670.802} C_VEL
LIN {X 0,Y 502.125,Z 498.733,A -85,B 0,C 180,E1 -5672.407,E2 -5672.407} C_VEL
LIN {X 0,Y 502.207,Z 497.385,A -85,B 0,C 180,E1 -5673.209,E2 -5673.209} C_VEL
LIN {X 0,Y 502.221,Z 494.546,A -85,B 0,C 180,E1 -5674.414,E2 -5674.414} C_VEL
LIN {X 0,Y 502.292,Z 490.692,A -85,B 0,C 180,E1 -5675.621,E2 -5675.621} C_VEL
LIN {X 0,Y 502.395,Z 485.718,A -85,B 0,C 180,E1 -5676.829,E2 -5676.829} C_VEL
LIN {X 0,Y 502.632,Z 479.447,A -85,B 0,C 180,E1 -5678.038,E2 -5678.038} C_VEL
LIN {X 0,Y 502.886,Z 471.595,A -85,B 0,C 180,E1 -5679.249,E2 -5679.249} C_VEL
LIN {X 0,Y 503.273,Z 461.817,A -85,B 0,C 180,E1 -5680.46,E2 -5680.46} C_VEL
LIN {X 0,Y 503.639,Z 451.556,A -85,B 0,C 180,E1 -5681.47,E2 -5681.47} C_VEL
LIN {X 0,Y 503.985,Z 439.842,A -85,B 0,C 180,E1 -5682.39,E2 -5682.39} C_VEL
LIN {X 0,Y 504.327,Z 428.441,A -85,B 0,C 180,E1 -5683.088,E2 -5683.088} C_VEL
LIN {X 0,Y 504.61,Z 416.44,A -85,B 0,C 180,E1 -5683.645,E2 -5683.645} C_VEL
LIN {X 0,Y 504.461,Z 408.671,A -85,B 0,C 180,E1 -5683.931,E2 -5683.931} C_VEL
LIN {X 0,Y 502.195,Z 397.747,A -85,B 0,C 180,E1 -5684.306,E2 -5684.306} C_VEL
LIN {X 0,Y 502.211,Z 393.529,A -85,B 0,C 180,E1 -5687.931,E2 -5687.931} C_VEL
LIN {X 0,Y 502.217,Z 390.666,A -85,B 0,C 180,E1 -5690.478,E2 -5690.478} C_VEL
LIN {X 0,Y 502.244,Z 387.912,A -85,B 0,C 180,E1 -5693.067,E2 -5693.067} C_VEL
LIN {X 0,Y 502.326,Z 385.168,A -85,B 0,C 180,E1 -5695.704,E2 -5695.704} C_VEL
LIN {X 0,Y 502.401,Z 382.44,A -85,B 0,C 180,E1 -5698.4,E2 -5698.4} C_VEL
LIN {X 0,Y 502.478,Z 379.384,A -85,B 0,C 180,E1 -5701.44,E2 -5701.44} C_VEL
LIN {X 0,Y 502.476,Z 377.897,A -85,B 0,C 180,E1 -5703.058,E2 -5703.058} C_VEL
LIN {X 0,Y 502.744,Z 377.861,A -85,B 0,C 180,E1 -5705.954,E2 -5705.954} C_VEL
LIN {X 0,Y 502.805,Z 377.854,A -85,B 0,C 180,E1 -5708.976,E2 -5708.976} C_VEL
LIN {X 0,Y 502.801,Z 377.856,A -85,B 0,C 180,E1 -5712.139,E2 -5712.139} C_VEL
LIN {X 0,Y 502.79,Z 377.856,A -85,B 0,C 180,E1 -5715.47,E2 -5715.47} C_VEL
LIN {X 0,Y 502.824,Z 377.853,A -85,B 0,C 180,E1 -5718.934,E2 -5718.934} C_VEL
LIN {X 0,Y 502.799,Z 377.854,A -85,B 0,C 180,E1 -5722.046,E2 -5722.046} C_VEL
LIN {X 0,Y 502.812,Z 377.85,A -85,B 0,C 180,E1 -5725.035,E2 -5725.035} C_VEL
LIN {X 0,Y 502.788,Z 377.858,A -85,B 0,C 180,E1 -5727.916,E2 -5727.916} C_VEL
LIN {X 0,Y 502.829,Z 377.852,A -85,B 0,C 180,E1 -5730.712,E2 -5730.712} C_VEL
LIN {X 0,Y 502.868,Z 377.845,A -85,B 0,C 180,E1 -5733.439,E2 -5733.439} C_VEL
LIN {X 0,Y 502.781,Z 377.86,A -85,B 0,C 180,E1 -5736.086,E2 -5736.086} C_VEL
LIN {X 0,Y 502.789,Z 377.853,A -85,B 0,C 180,E1 -5738.689,E2 -5738.689} C_VEL
LIN {X 0,Y 502.833,Z 377.851,A -85,B 0,C 180,E1 -5741.248,E2 -5741.248} C_VEL
LIN {X 0,Y 502.854,Z 377.849,A -85,B 0,C 180,E1 -5744.6,E2 -5744.6} C_VEL
LIN {X 0,Y 502.882,Z 377.848,A -85,B 0,C 180,E1 -5748.039,E2 -5748.039} C_VEL
LIN {X 0,Y 502.87,Z 377.844,A -85,B 0,C 180,E1 -5751.157,E2 -5751.157} C_VEL
LIN {X 0,Y 502.933,Z 377.839,A -85,B 0,C 180,E1 -5753.581,E2 -5753.581} C_VEL
LIN {X 0,Y 503.028,Z 377.825,A -85,B 0,C 180,E1 -5757.598,E2 -5757.598} C_VEL
LIN {X 0,Y 503.033,Z 377.829,A -85,B 0,C 180,E1 -5760,E2 -5760} C_VEL
LIN {X 0,Y 503.03,Z 377.823,A -85,B 0,C 180,E1 -5762.402,E2 -5762.402} C_VEL
LIN {X 0,Y 502.933,Z 377.837,A -85,B 0,C 180,E1 -5766.419,E2 -5766.419} C_VEL
LIN {X 0,Y 502.88,Z 377.846,A -85,B 0,C 180,E1 -5768.843,E2 -5768.843} C_VEL
LIN {X 0,Y 502.899,Z 377.843,A -85,B 0,C 180,E1 -5772.1,E2 -5772.1} C_VEL
LIN {X 0,Y 502.854,Z 377.85,A -85,B 0,C 180,E1 -5775.4,E2 -5775.4} C_VEL
LIN {X 0,Y 502.832,Z 377.851,A -85,B 0,C 180,E1 -5778.752,E2 -5778.752} C_VEL
LIN {X 0,Y 502.789,Z 377.855,A -85,B 0,C 180,E1 -5781.311,E2 -5781.311} C_VEL
LIN {X 0,Y 502.781,Z 377.859,A -85,B 0,C 180,E1 -5783.914,E2 -5783.914} C_VEL
LIN {X 0,Y 502.869,Z 377.844,A -85,B 0,C 180,E1 -5786.566,E2 -5786.566} C_VEL
LIN {X 0,Y 502.829,Z 377.853,A -85,B 0,C 180,E1 -5789.288,E2 -5789.288} C_VEL
LIN {X 0,Y 502.788,Z 377.855,A -85,B 0,C 180,E1 -5792.084,E2 -5792.084} C_VEL
LIN {X 0,Y 502.803,Z 377.853,A -85,B 0,C 180,E1 -5794.966,E2 -5794.966} C_VEL
LIN {X 0,Y 502.798,Z 377.855,A -85,B 0,C 180,E1 -5797.954,E2 -5797.954} C_VEL
LIN {X 0,Y 502.823,Z 377.854,A -85,B 0,C 180,E1 -5801.066,E2 -5801.066} C_VEL
LIN {X 0,Y 502.805,Z 377.856,A -85,B 0,C 180,E1 -5804.532,E2 -5804.532} C_VEL
LIN {X 0,Y 502.834,Z 377.853,A -85,B 0,C 180,E1 -5807.864,E2 -5807.864} C_VEL
LIN {X 0,Y 502.82,Z 377.918,A -85,B 0,C 180,E1 -5810.896,E2 -5810.896} C_VEL
LIN {X 0,Y 504.012,Z 384.68,A -85,B 0,C 180,E1 -5813.6,E2 -5813.6} C_VEL
LIN {X 0,Y 504.126,Z 389.447,A -85,B 0,C 180,E1 -5815.338,E2 -5815.338} C_VEL
LIN {X 0,Y 503.876,Z 397.914,A -85,B 0,C 180,E1 -5818.301,E2 -5818.301} C_VEL
LIN {X 0,Y 503.585,Z 406.488,A -85,B 0,C 180,E1 -5821.203,E2 -5821.203} C_VEL
LIN {X 0,Y 503.331,Z 414.728,A -85,B 0,C 180,E1 -5823.906,E2 -5823.906} C_VEL
LIN {X 0,Y 503.141,Z 422.9,A -85,B 0,C 180,E1 -5826.541,E2 -5826.541} C_VEL
LIN {X 0,Y 502.903,Z 432.167,A -85,B 0,C 180,E1 -5829.551,E2 -5829.551} C_VEL
LIN {X 0,Y 502.664,Z 441.435,A -85,B 0,C 180,E1 -5832.506,E2 -5832.506} C_VEL
LIN {X 0,Y 502.506,Z 451.581,A -85,B 0,C 180,E1 -5835.694,E2 -5835.694} C_VEL
LIN {X 0,Y 504.69,Z 465.089,A -85,B 0,C 180,E1 -5836.075,E2 -5836.075} C_VEL
LIN {X 0,Y 504.428,Z 478.108,A -85,B 0,C 180,E1 -5836.555,E2 -5836.555} C_VEL
LIN {X 0,Y 504.055,Z 490.528,A -85,B 0,C 180,E1 -5837.188,E2 -5837.188} C_VEL
LIN {X 0,Y 503.741,Z 501.586,A -85,B 0,C 180,E1 -5837.92,E2 -5837.92} C_VEL
LIN {X 0,Y 503.385,Z 512.467,A -85,B 0,C 180,E1 -5838.83,E2 -5838.83} C_VEL
LIN {X 0,Y 503.024,Z 521.332,A -85,B 0,C 180,E1 -5839.739,E2 -5839.739} C_VEL
LIN {X 0,Y 502.704,Z 530.96,A -85,B 0,C 180,E1 -5840.951,E2 -5840.951} C_VEL
LIN {X 0,Y 502.47,Z 538.621,A -85,B 0,C 180,E1 -5842.162,E2 -5842.162} C_VEL
LIN {X 0,Y 502.275,Z 545.679,A -85,B 0,C 180,E1 -5843.573,E2 -5843.573} C_VEL
LIN {X 0,Y 502.186,Z 550.372,A -85,B 0,C 180,E1 -5844.781,E2 -5844.781} C_VEL
LIN {X 0,Y 502.151,Z 553.958,A -85,B 0,C 180,E1 -5845.987,E2 -5845.987} C_VEL
LIN {X 0,Y 502.121,Z 555.807,A -85,B 0,C 180,E1 -5846.79,E2 -5846.79} C_VEL
LIN {X 0,Y 502.066,Z 557.195,A -85,B 0,C 180,E1 -5847.593,E2 -5847.593} C_VEL
LIN {X 0,Y 501.99,Z 558.786,A -85,B 0,C 180,E1 -5849.198,E2 -5849.198} C_VEL
LIN {X 0,Y 501.98,Z 559,A -85,B 0,C 180,E1 -5850,E2 -5850} C_VEL
LIN {X 0,Y 502.036,Z 558.185,A -85,B 0,C 180,E1 -5851.604,E2 -5851.604} C_VEL
LIN {X 0,Y 502.066,Z 557.198,A -85,B 0,C 180,E1 -5852.407,E2 -5852.407} C_VEL
LIN {X 0,Y 502.121,Z 555.81,A -85,B 0,C 180,E1 -5853.209,E2 -5853.209} C_VEL
LIN {X 0,Y 502.128,Z 552.896,A -85,B 0,C 180,E1 -5854.415,E2 -5854.415} C_VEL
LIN {X 0,Y 502.259,Z 548.949,A -85,B 0,C 180,E1 -5855.621,E2 -5855.621} C_VEL
LIN {X 0,Y 502.336,Z 542.977,A -85,B 0,C 180,E1 -5857.011,E2 -5857.011} C_VEL
LIN {X 0,Y 502.542,Z 536.236,A -85,B 0,C 180,E1 -5858.241,E2 -5858.241} C_VEL
LIN {X 0,Y 502.811,Z 527.991,A -85,B 0,C 180,E1 -5859.453,E2 -5859.453} C_VEL
LIN {X 0,Y 503.065,Z 519.539,A -85,B 0,C 180,E1 -5860.464,E2 -5860.464} C_VEL
LIN {X 0,Y 503.532,Z 509.094,A -85,B 0,C 180,E1 -5861.472,E2 -5861.472} C_VEL
LIN {X 0,Y 503.805,Z 497.501,A -85,B 0,C 180,E1 -5862.372,E2 -5862.372} C_VEL
LIN {X 0,Y 504.216,Z 485.489,A -85,B 0,C 180,E1 -5863.091,E2 -5863.091} C_VEL
LIN {X 0,Y 504.533,Z 473.166,A -85,B 0,C 180,E1 -5863.647,E2 -5863.647} C_VEL
LIN {X 0,Y 504.506,Z 463.717,A -85,B 0,C 180,E1 -5863.969,E2 -5863.969} C_VEL
LIN {X 0,Y 502.505,Z 451.53,A -85,B 0,C 180,E1 -5864.322,E2 -5864.322} C_VEL
LIN {X 0,Y 502.664,Z 441.435,A -85,B 0,C 180,E1 -5867.494,E2 -5867.494} C_VEL
LIN {X 0,Y 502.907,Z 431.827,A -85,B 0,C 180,E1 -5870.559,E2 -5870.559} C_VEL
LIN {X 0,Y 503.189,Z 421.577,A -85,B 0,C 180,E1 -5873.894,E2 -5873.894} C_VEL
LIN {X 0,Y 503.455,Z 411.904,A -85,B 0,C 180,E1 -5877.012,E2 -5877.012} C_VEL
LIN {X 0,Y 503.724,Z 402.43,A -85,B 0,C 180,E1 -5880.151,E2 -5880.151} C_VEL
LIN {X 0,Y 504.033,Z 393.547,A -85,B 0,C 180,E1 -5883.216,E2 -5883.216} C_VEL
LIN {X 0,Y 504.186,Z 386.177,A -85,B 0,C 180,E1 -5885.835,E2 -5885.835} C_VEL
LIN {X 0,Y 503.346,Z 380.852,A -85,B 0,C 180,E1 -5887.905,E2 -5887.905} C_VEL
LIN {X 0,Y 502.808,Z 377.856,A -85,B 0,C 180,E1 -5889.169,E2 -5889.169} C_VEL
LIN {X 0,Y 502.806,Z 377.859,A -85,B 0,C 180,E1 -5892.199,E2 -5892.199} C_VEL
LIN {X 0,Y 502.804,Z 377.861,A -85,B 0,C 180,E1 -5895.468,E2 -5895.468} C_VEL
LIN {X 0,Y 502.823,Z 377.855,A -85,B 0,C 180,E1 -5898.934,E2 -5898.934} C_VEL
LIN {X 0,Y 502.797,Z 377.855,A -85,B 0,C 180,E1 -5902.046,E2 -5902.046} C_VEL
LIN {X 0,Y 502.81,Z 377.853,A -85,B 0,C 180,E1 -5905.035,E2 -5905.035} C_VEL
LIN {X 0,Y 502.786,Z 377.855,A -85,B 0,C 180,E1 -5907.916,E2 -5907.916} C_VEL
LIN {X 0,Y 502.828,Z 377.853,A -85,B 0,C 180,E1 -5910.712,E2 -5910.712} C_VEL
LIN {X 0,Y 502.866,Z 377.844,A -85,B 0,C 180,E1 -5913.439,E2 -5913.439} C_VEL
LIN {X 0,Y 502.78,Z 377.859,A -85,B 0,C 180,E1 -5916.086,E2 -5916.086} C_VEL
LIN {X 0,Y 502.787,Z 377.855,A -85,B 0,C 180,E1 -5918.689,E2 -5918.689} C_VEL
LIN {X 0,Y 502.834,Z 377.85,A -85,B 0,C 180,E1 -5921.248,E2 -5921.248} C_VEL
LIN {X 0,Y 502.826,Z 377.848,A -85,B 0,C 180,E1 -5923.767,E2 -5923.767} C_VEL
LIN {X 0,Y 502.836,Z 377.852,A -85,B 0,C 180,E1 -5926.255,E2 -5926.255} C_VEL
LIN {X 0,Y 502.896,Z 377.841,A -85,B 0,C 180,E1 -5928.717,E2 -5928.717} C_VEL
LIN {X 0,Y 502.906,Z 377.841,A -85,B 0,C 180,E1 -5931.967,E2 -5931.967} C_VEL
LIN {X 0,Y 502.941,Z 377.837,A -85,B 0,C 180,E1 -5934.387,E2 -5934.387} C_VEL
LIN {X 0,Y 503.028,Z 377.823,A -85,B 0,C 180,E1 -5937.598,E2 -5937.598} C_VEL
LIN {X 0,Y 503.031,Z 377.828,A -85,B 0,C 180,E1 -5940,E2 -5940} C_VEL
LIN {X 0,Y 503.026,Z 377.825,A -85,B 0,C 180,E1 -5942.402,E2 -5942.402} C_VEL
LIN {X 0,Y 502.942,Z 377.836,A -85,B 0,C 180,E1 -5945.614,E2 -5945.614} C_VEL
LIN {X 0,Y 502.904,Z 377.841,A -85,B 0,C 180,E1 -5948.033,E2 -5948.033} C_VEL
LIN {X 0,Y 502.881,Z 377.842,A -85,B 0,C 180,E1 -5951.283,E2 -5951.283} C_VEL
LIN {X 0,Y 502.849,Z 377.847,A -85,B 0,C 180,E1 -5954.571,E2 -5954.571} C_VEL
LIN {X 0,Y 502.827,Z 377.85,A -85,B 0,C 180,E1 -5957.908,E2 -5957.908} C_VEL
LIN {X 0,Y 502.833,Z 377.851,A -85,B 0,C 180,E1 -5960.536,E2 -5960.536} C_VEL
LIN {X 0,Y 502.792,Z 377.852,A -85,B 0,C 180,E1 -5963.041,E2 -5963.041} C_VEL
LIN {X 0,Y 502.826,Z 377.854,A -85,B 0,C 180,E1 -5965.677,E2 -5965.677} C_VEL
LIN {X 0,Y 502.844,Z 377.848,A -85,B 0,C 180,E1 -5968.373,E2 -5968.373} C_VEL
LIN {X 0,Y 502.796,Z 377.854,A -85,B 0,C 180,E1 -5971.499,E2 -5971.499} C_VEL
LIN {X 0,Y 502.808,Z 377.856,A -85,B 0,C 180,E1 -5973.994,E2 -5973.994} C_VEL
LIN {X 0,Y 502.781,Z 377.855,A -85,B 0,C 180,E1 -5977.178,E2 -5977.178} C_VEL
LIN {X 0,Y 502.792,Z 377.854,A -85,B 0,C 180,E1 -5980.015,E2 -5980.015} C_VEL
LIN {X 0,Y 502.806,Z 377.854,A -85,B 0,C 180,E1 -5982.199,E2 -5982.199} C_VEL
LIN {X 0,Y 502.789,Z 377.855,A -85,B 0,C 180,E1 -5985.47,E2 -5985.47} C_VEL
LIN {X 0,Y 502.833,Z 377.853,A -85,B 0,C 180,E1 -5987.864,E2 -5987.864} C_VEL
LIN {X 0,Y 502.804,Z 377.853,A -85,B 0,C 180,E1 -5991.024,E2 -5991.024} C_VEL
LIN {X 0,Y 502.742,Z 377.862,A -85,B 0,C 180,E1 -5994.175,E2 -5994.175} C_VEL
LIN {X 0,Y 502.475,Z 377.898,A -85,B 0,C 180,E1 -5997.057,E2 -5997.057} C_VEL
LIN {X 0,Y 502.465,Z 378.038,A -85,B 0,C 180,E1 -5997.215,E2 -5997.215} C_VEL
LIN {X 0,Y 501.775,Z 378.714,A -85,B 0,C 180,E1 -5997.88,E2 -5997.88} C_VEL
LIN {X 0,Y 498.893,Z 380.049,A -85,B 0,C 180,E1 -5998.955,E2 -5998.955} C_VEL
LIN {X 0,Y 496.461,Z 381.154,A -85,B 0,C 180,E1 -5999.821,E2 -5999.821} C_VEL
LIN {X 0,Y 495.411,Z 381.928,A -85,B 0,C 180,E1 -6000.491,E2 -6000.491} C_VEL
LIN {X 0,Y 495.322,Z 382.165,A -85,B 0,C 180,E1 -6000.719,E2 -6000.719} C_VEL
LIN {X 0,Y 495.281,Z 384.855,A -85,B 0,C 180,E1 -6003.376,E2 -6003.376} C_VEL
LIN {X 0,Y 495.223,Z 387.215,A -85,B 0,C 180,E1 -6005.697,E2 -6005.697} C_VEL
LIN {X 0,Y 495.157,Z 389.95,A -85,B 0,C 180,E1 -6008.344,E2 -6008.344} C_VEL
LIN {X 0,Y 495.13,Z 392.759,A -85,B 0,C 180,E1 -6010.945,E2 -6010.945} C_VEL
LIN {X 0,Y 495.09,Z 395.67,A -85,B 0,C 180,E1 -6013.506,E2 -6013.506} C_VEL
LIN {X 0,Y 495.141,Z 398.187,A -85,B 0,C 180,E1 -6015.591,E2 -6015.591} C_VEL
LIN {X 0,Y 497.688,Z 410.246,A -85,B 0,C 180,E1 -6016.006,E2 -6016.006} C_VEL
LIN {X 0,Y 497.597,Z 423.05,A -85,B 0,C 180,E1 -6016.524,E2 -6016.524} C_VEL
LIN {X 0,Y 497.303,Z 434.502,A -85,B 0,C 180,E1 -6017.145,E2 -6017.145} C_VEL
LIN {X 0,Y 496.889,Z 446.054,A -85,B 0,C 180,E1 -6017.958,E2 -6017.958} C_VEL
LIN {X 0,Y 496.526,Z 456.486,A -85,B 0,C 180,E1 -6018.881,E2 -6018.881} C_VEL
LIN {X 0,Y 496.187,Z 465.006,A -85,B 0,C 180,E1 -6019.802,E2 -6019.802} C_VEL
LIN {X 0,Y 495.898,Z 472.847,A -85,B 0,C 180,E1 -6020.826,E2 -6020.826} C_VEL
LIN {X 0,Y 495.579,Z 480.514,A -85,B 0,C 180,E1 -6022.052,E2 -6022.052} C_VEL
LIN {X 0,Y 495.341,Z 487.537,A -85,B 0,C 180,E1 -6023.483,E2 -6023.483} C_VEL
LIN {X 0,Y 495.135,Z 492.22,A -85,B 0,C 180,E1 -6024.706,E2 -6024.706} C_VEL
LIN {X 0,Y 495.173,Z 495.794,A -85,B 0,C 180,E1 -6025.931,E2 -6025.931} C_VEL
LIN {X 0,Y 495.139,Z 497.644,A -85,B 0,C 180,E1 -6026.745,E2 -6026.745} C_VEL
LIN {X 0,Y 495.061,Z 499.043,A -85,B 0,C 180,E1 -6027.559,E2 -6027.559} C_VEL
LIN {X 0,Y 494.915,Z 500.654,A -85,B 0,C 180,E1 -6029.186,E2 -6029.186} C_VEL
LIN {X 0,Y 494.906,Z 500.889,A -85,B 0,C 180,E1 -6030,E2 -6030} C_VEL
LIN {X 0,Y 494.915,Z 500.705,A -85,B 0,C 180,E1 -6030.814,E2 -6030.814} C_VEL
LIN {X 0,Y 495.061,Z 499.162,A -85,B 0,C 180,E1 -6032.441,E2 -6032.441} C_VEL
LIN {X 0,Y 495.139,Z 497.815,A -85,B 0,C 180,E1 -6033.255,E2 -6033.255} C_VEL
LIN {X 0,Y 495.154,Z 494.976,A -85,B 0,C 180,E1 -6034.477,E2 -6034.477} C_VEL
LIN {X 0,Y 495.24,Z 491.121,A -85,B 0,C 180,E1 -6035.701,E2 -6035.701} C_VEL
LIN {X 0,Y 495.364,Z 486.147,A -85,B 0,C 180,E1 -6036.926,E2 -6036.926} C_VEL
LIN {X 0,Y 495.622,Z 479.874,A -85,B 0,C 180,E1 -6038.152,E2 -6038.152} C_VEL
LIN {X 0,Y 495.885,Z 472.022,A -85,B 0,C 180,E1 -6039.38,E2 -6039.38} C_VEL
LIN {X 0,Y 496.314,Z 462.243,A -85,B 0,C 180,E1 -6040.608,E2 -6040.608} C_VEL
LIN {X 0,Y 496.712,Z 451.979,A -85,B 0,C 180,E1 -6041.632,E2 -6041.632} C_VEL
LIN {X 0,Y 497.073,Z 440.635,A -85,B 0,C 180,E1 -6042.538,E2 -6042.538} C_VEL
LIN {X 0,Y 497.427,Z 428.86,A -85,B 0,C 180,E1 -6043.273,E2 -6043.273} C_VEL
LIN {X 0,Y 497.746,Z 416.854,A -85,B 0,C 180,E1 -6043.837,E2 -6043.837} C_VEL
LIN {X 0,Y 497.606,Z 409.841,A -85,B 0,C 180,E1 -6044.101,E2 -6044.101} C_VEL
LIN {X 0,Y 495.114,Z 398.115,A -85,B 0,C 180,E1 -6044.515,E2 -6044.515} C_VEL
LIN {X 0,Y 495.131,Z 394.797,A -85,B 0,C 180,E1 -6047.342,E2 -6047.342} C_VEL
LIN {X 0,Y 495.137,Z 390.964,A -85,B 0,C 180,E1 -6050.785,E2 -6050.785} C_VEL
LIN {X 0,Y 495.187,Z 388.203,A -85,B 0,C 180,E1 -6053.416,E2 -6053.416} C_VEL
LIN {X 0,Y 495.268,Z 385.439,A -85,B 0,C 180,E1 -6056.098,E2 -6056.098} C_VEL
LIN {X 0,Y 495.32,Z 382.69,A -85,B 0,C 180,E1 -6058.844,E2 -6058.844} C_VEL
LIN {X 0,Y 495.415,Z 379.875,A -85,B 0,C 180,E1 -6061.661,E2 -6061.661} C_VEL
LIN {X 0,Y 495.394,Z 378.927,A -85,B 0,C 180,E1 -6062.622,E2 -6062.622} C_VEL
LIN {X 0,Y 495.668,Z 378.743,A -85,B 0,C 180,E1 -6065.545,E2 -6065.545} C_VEL
LIN {X 0,Y 495.767,Z 378.733,A -85,B 0,C 180,E1 -6068.768,E2 -6068.768} C_VEL
LIN {X 0,Y 495.761,Z 378.729,A -85,B 0,C 180,E1 -6071.781,E2 -6071.781} C_VEL
LIN {X 0,Y 495.741,Z 378.734,A -85,B 0,C 180,E1 -6075.141,E2 -6075.141} C_VEL
LIN {X 0,Y 495.76,Z 378.731,A -85,B 0,C 180,E1 -6078.219,E2 -6078.219} C_VEL
LIN {X 0,Y 495.756,Z 378.73,A -85,B 0,C 180,E1 -6081.409,E2 -6081.409} C_VEL
LIN {X 0,Y 495.76,Z 378.732,A -85,B 0,C 180,E1 -6084.463,E2 -6084.463} C_VEL
LIN {X 0,Y 495.772,Z 378.73,A -85,B 0,C 180,E1 -6087.406,E2 -6087.406} C_VEL
LIN {X 0,Y 495.771,Z 378.729,A -85,B 0,C 180,E1 -6090.254,E2 -6090.254} C_VEL
LIN {X 0,Y 495.828,Z 378.723,A -85,B 0,C 180,E1 -6093.251,E2 -6093.251} C_VEL
LIN {X 0,Y 495.748,Z 378.731,A -85,B 0,C 180,E1 -6096.613,E2 -6096.613} C_VEL
LIN {X 0,Y 495.784,Z 378.728,A -85,B 0,C 180,E1 -6099.324,E2 -6099.324} C_VEL
LIN {X 0,Y 495.787,Z 378.728,A -85,B 0,C 180,E1 -6101.829,E2 -6101.829} C_VEL
LIN {X 0,Y 495.829,Z 378.724,A -85,B 0,C 180,E1 -6104.548,E2 -6104.548} C_VEL
LIN {X 0,Y 495.834,Z 378.725,A -85,B 0,C 180,E1 -6107.965,E2 -6107.965} C_VEL
LIN {X 0,Y 495.84,Z 378.719,A -85,B 0,C 180,E1 -6111.03,E2 -6111.03} C_VEL
LIN {X 0,Y 495.885,Z 378.718,A -85,B 0,C 180,E1 -6113.49,E2 -6113.49} C_VEL
LIN {X 0,Y 495.844,Z 378.721,A -85,B 0,C 180,E1 -6116.75,E2 -6116.75} C_VEL
LIN {X 0,Y 495.875,Z 378.718,A -85,B 0,C 180,E1 -6118.376,E2 -6118.376} C_VEL
LIN {X 0,Y 495.989,Z 378.701,A -85,B 0,C 180,E1 -6120.812,E2 -6120.812} C_VEL
LIN {X 0,Y 495.998,Z 378.698,A -85,B 0,C 180,E1 -6122.436,E2 -6122.436} C_VEL
LIN {X 0,Y 495.9,Z 378.714,A -85,B 0,C 180,E1 -6125.693,E2 -6125.693} C_VEL
LIN {X 0,Y 495.879,Z 378.717,A -85,B 0,C 180,E1 -6128.148,E2 -6128.148} C_VEL
LIN {X 0,Y 495.873,Z 378.717,A -85,B 0,C 180,E1 -6131.445,E2 -6131.445} C_VEL
LIN {X 0,Y 495.796,Z 378.724,A -85,B 0,C 180,E1 -6134.783,E2 -6134.783} C_VEL
LIN {X 0,Y 495.769,Z 378.733,A -85,B 0,C 180,E1 -6137.319,E2 -6137.319} C_VEL
LIN {X 0,Y 495.783,Z 378.727,A -85,B 0,C 180,E1 -6139.89,E2 -6139.89} C_VEL
LIN {X 0,Y 495.764,Z 378.731,A -85,B 0,C 180,E1 -6142.86,E2 -6142.86} C_VEL
LIN {X 0,Y 495.785,Z 378.728,A -85,B 0,C 180,E1 -6146.068,E2 -6146.068} C_VEL
LIN {X 0,Y 495.777,Z 378.728,A -85,B 0,C 180,E1 -6148.815,E2 -6148.815} C_VEL
LIN {X 0,Y 495.76,Z 378.73,A -85,B 0,C 180,E1 -6151.725,E2 -6151.725} C_VEL
LIN {X 0,Y 495.773,Z 378.731,A -85,B 0,C 180,E1 -6154.694,E2 -6154.694} C_VEL
LIN {X 0,Y 495.734,Z 378.737,A -85,B 0,C 180,E1 -6157.561,E2 -6157.561} C_VEL
LIN {X 0,Y 495.77,Z 378.729,A -85,B 0,C 180,E1 -6160.7,E2 -6160.7} C_VEL
LIN {X 0,Y 495.738,Z 378.734,A -85,B 0,C 180,E1 -6164.001,E2 -6164.001} C_VEL
LIN {X 0,Y 495.738,Z 378.735,A -85,B 0,C 180,E1 -6167.118,E2 -6167.118} C_VEL
LIN {X 0,Y 495.762,Z 378.733,A -85,B 0,C 180,E1 -6169.953,E2 -6169.953} C_VEL
LIN {X 0,Y 495.779,Z 378.84,A -85,B 0,C 180,E1 -6170.646,E2 -6170.646} C_VEL
LIN {X 0,Y 497.043,Z 386.005,A -85,B 0,C 180,E1 -6173.568,E2 -6173.568} C_VEL
LIN {X 0,Y 497.127,Z 391.407,A -85,B 0,C 180,E1 -6175.563,E2 -6175.563} C_VEL
LIN {X 0,Y 496.835,Z 399.535,A -85,B 0,C 180,E1 -6178.44,E2 -6178.44} C_VEL
LIN {X 0,Y 496.56,Z 408.02,A -85,B 0,C 180,E1 -6181.344,E2 -6181.344} C_VEL
LIN {X 0,Y 496.311,Z 415.87,A -85,B 0,C 180,E1 -6183.961,E2 -6183.961} C_VEL
LIN {X 0,Y 496.094,Z 424.074,A -85,B 0,C 180,E1 -6186.63,E2 -6186.63} C_VEL
LIN {X 0,Y 495.843,Z 433.553,A -85,B 0,C 180,E1 -6189.7,E2 -6189.7} C_VEL
LIN {X 0,Y 495.594,Z 442.759,A -85,B 0,C 180,E1 -6192.674,E2 -6192.674} C_VEL
LIN {X 0,Y 495.433,Z 451.581,A -85,B 0,C 180,E1 -6195.485,E2 -6195.485} C_VEL
LIN {X 0,Y 497.704,Z 465.089,A -85,B 0,C 180,E1 -6195.876,E2 -6195.876} C_VEL
LIN {X 0,Y 497.516,Z 478.107,A -85,B 0,C 180,E1 -6196.365,E2 -6196.365} C_VEL
LIN {X 0,Y 497.129,Z 490.667,A -85,B 0,C 180,E1 -6197.015,E2 -6197.015} C_VEL
LIN {X 0,Y 496.782,Z 501.586,A -85,B 0,C 180,E1 -6197.748,E2 -6197.748} C_VEL
LIN {X 0,Y 496.411,Z 512.467,A -85,B 0,C 180,E1 -6198.671,E2 -6198.671} C_VEL
LIN {X 0,Y 495.998,Z 521.332,A -85,B 0,C 180,E1 -6199.592,E2 -6199.592} C_VEL
LIN {X 0,Y 495.673,Z 530.96,A -85,B 0,C 180,E1 -6200.821,E2 -6200.821} C_VEL
LIN {X 0,Y 495.404,Z 538.621,A -85,B 0,C 180,E1 -6202.049,E2 -6202.049} C_VEL
LIN {X 0,Y 495.204,Z 545.679,A -85,B 0,C 180,E1 -6203.481,E2 -6203.481} C_VEL
LIN {X 0,Y 495.123,Z 550.372,A -85,B 0,C 180,E1 -6204.706,E2 -6204.706} C_VEL
LIN {X 0,Y 495.049,Z 553.958,A -85,B 0,C 180,E1 -6205.929,E2 -6205.929} C_VEL
LIN {X 0,Y 495.043,Z 555.807,A -85,B 0,C 180,E1 -6206.744,E2 -6206.744} C_VEL
LIN {X 0,Y 494.961,Z 558.183,A -85,B 0,C 180,E1 -6208.373,E2 -6208.373} C_VEL
LIN {X 0,Y 494.898,Z 559,A -85,B 0,C 180,E1 -6210,E2 -6210} C_VEL
LIN {X 0,Y 494.961,Z 558.185,A -85,B 0,C 180,E1 -6211.627,E2 -6211.627} C_VEL
LIN {X 0,Y 495.043,Z 555.81,A -85,B 0,C 180,E1 -6213.255,E2 -6213.255} C_VEL
LIN {X 0,Y 495.029,Z 552.896,A -85,B 0,C 180,E1 -6214.478,E2 -6214.478} C_VEL
LIN {X 0,Y 495.209,Z 547.804,A -85,B 0,C 180,E1 -6215.999,E2 -6215.999} C_VEL
LIN {X 0,Y 495.277,Z 541.869,A -85,B 0,C 180,E1 -6217.337,E2 -6217.337} C_VEL
LIN {X 0,Y 495.557,Z 535.003,A -85,B 0,C 180,E1 -6218.564,E2 -6218.564} C_VEL
LIN {X 0,Y 495.847,Z 526.413,A -85,B 0,C 180,E1 -6219.793,E2 -6219.793} C_VEL
LIN {X 0,Y 496.188,Z 517.599,A -85,B 0,C 180,E1 -6220.817,E2 -6220.817} C_VEL
LIN {X 0,Y 496.622,Z 506.744,A -85,B 0,C 180,E1 -6221.841,E2 -6221.841} C_VEL
LIN {X 0,Y 496.902,Z 496.738,A -85,B 0,C 180,E1 -6222.601,E2 -6222.601} C_VEL
LIN {X 0,Y 497.298,Z 485.488,A -85,B 0,C 180,E1 -6223.277,E2 -6223.277} C_VEL
LIN {X 0,Y 497.65,Z 473.165,A -85,B 0,C 180,E1 -6223.839,E2 -6223.839} C_VEL
LIN {X 0,Y 497.621,Z 464.63,A -85,B 0,C 180,E1 -6224.14,E2 -6224.14} C_VEL
LIN {X 0,Y 495.443,Z 451.53,A -85,B 0,C 180,E1 -6224.531,E2 -6224.531} C_VEL
LIN {X 0,Y 495.639,Z 441.435,A -85,B 0,C 180,E1 -6227.75,E2 -6227.75} C_VEL
LIN {X 0,Y 495.887,Z 432.168,A -85,B 0,C 180,E1 -6230.752,E2 -6230.752} C_VEL
LIN {X 0,Y 496.121,Z 422.7,A -85,B 0,C 180,E1 -6233.811,E2 -6233.811} C_VEL
LIN {X 0,Y 496.418,Z 413.128,A -85,B 0,C 180,E1 -6236.939,E2 -6236.939} C_VEL
LIN {X 0,Y 496.738,Z 403.042,A -85,B 0,C 180,E1 -6240.339,E2 -6240.339} C_VEL
LIN {X 0,Y 497.056,Z 394.124,A -85,B 0,C 180,E1 -6243.465,E2 -6243.465} C_VEL
LIN {X 0,Y 497.213,Z 387.517,A -85,B 0,C 180,E1 -6245.854,E2 -6245.854} C_VEL
LIN {X 0,Y 496.35,Z 382.049,A -85,B 0,C 180,E1 -6248.019,E2 -6248.019} C_VEL
LIN {X 0,Y 495.751,Z 378.735,A -85,B 0,C 180,E1 -6249.412,E2 -6249.412} C_VEL
LIN {X 0,Y 495.744,Z 378.737,A -85,B 0,C 180,E1 -6252.507,E2 -6252.507} C_VEL
LIN {X 0,Y 495.752,Z 378.739,A -85,B 0,C 180,E1 -6255.139,E2 -6255.139} C_VEL
LIN {X 0,Y 495.759,Z 378.728,A -85,B 0,C 180,E1 -6258.219,E2 -6258.219} C_VEL
LIN {X 0,Y 495.754,Z 378.731,A -85,B 0,C 180,E1 -6261.409,E2 -6261.409} C_VEL
LIN {X 0,Y 495.758,Z 378.732,A -85,B 0,C 180,E1 -6264.463,E2 -6264.463} C_VEL
LIN {X 0,Y 495.771,Z 378.731,A -85,B 0,C 180,E1 -6267.406,E2 -6267.406} C_VEL
LIN {X 0,Y 495.77,Z 378.728,A -85,B 0,C 180,E1 -6270.254,E2 -6270.254} C_VEL
LIN {X 0,Y 495.827,Z 378.721,A -85,B 0,C 180,E1 -6273.251,E2 -6273.251} C_VEL
LIN {X 0,Y 495.746,Z 378.733,A -85,B 0,C 180,E1 -6276.613,E2 -6276.613} C_VEL
LIN {X 0,Y 495.782,Z 378.73,A -85,B 0,C 180,E1 -6279.324,E2 -6279.324} C_VEL
LIN {X 0,Y 495.802,Z 378.724,A -85,B 0,C 180,E1 -6281.829,E2 -6281.829} C_VEL
LIN {X 0,Y 495.828,Z 378.727,A -85,B 0,C 180,E1 -6284.548,E2 -6284.548} C_VEL
LIN {X 0,Y 495.881,Z 378.717,A -85,B 0,C 180,E1 -6287.939,E2 -6287.939} C_VEL
LIN {X 0,Y 495.847,Z 378.722,A -85,B 0,C 180,E1 -6291.03,E2 -6291.03} C_VEL
LIN {X 0,Y 495.883,Z 378.716,A -85,B 0,C 180,E1 -6293.49,E2 -6293.49} C_VEL
LIN {X 0,Y 495.845,Z 378.721,A -85,B 0,C 180,E1 -6296.75,E2 -6296.75} C_VEL
LIN {X 0,Y 496.009,Z 378.698,A -85,B 0,C 180,E1 -6299.188,E2 -6299.188} C_VEL
LIN {X 0,Y 495.874,Z 378.718,A -85,B 0,C 180,E1 -6301.624,E2 -6301.624} C_VEL
LIN {X 0,Y 495.844,Z 378.721,A -85,B 0,C 180,E1 -6303.25,E2 -6303.25} C_VEL
LIN {X 0,Y 495.884,Z 378.718,A -85,B 0,C 180,E1 -6306.51,E2 -6306.51} C_VEL
LIN {X 0,Y 495.841,Z 378.719,A -85,B 0,C 180,E1 -6308.97,E2 -6308.97} C_VEL
LIN {X 0,Y 495.832,Z 378.725,A -85,B 0,C 180,E1 -6312.035,E2 -6312.035} C_VEL
LIN {X 0,Y 495.828,Z 378.724,A -85,B 0,C 180,E1 -6315.452,E2 -6315.452} C_VEL
LIN {X 0,Y 495.783,Z 378.729,A -85,B 0,C 180,E1 -6318.237,E2 -6318.237} C_VEL
LIN {X 0,Y 495.778,Z 378.728,A -85,B 0,C 180,E1 -6320.756,E2 -6320.756} C_VEL
LIN {X 0,Y 495.747,Z 378.73,A -85,B 0,C 180,E1 -6323.387,E2 -6323.387} C_VEL
LIN {X 0,Y 495.827,Z 378.722,A -85,B 0,C 180,E1 -6326.749,E2 -6326.749} C_VEL
LIN {X 0,Y 495.77,Z 378.73,A -85,B 0,C 180,E1 -6329.746,E2 -6329.746} C_VEL
LIN {X 0,Y 495.771,Z 378.73,A -85,B 0,C 180,E1 -6332.594,E2 -6332.594} C_VEL
LIN {X 0,Y 495.751,Z 378.732,A -85,B 0,C 180,E1 -6335.538,E2 -6335.538} C_VEL
LIN {X 0,Y 495.768,Z 378.729,A -85,B 0,C 180,E1 -6338.768,E2 -6338.768} C_VEL
LIN {X 0,Y 495.76,Z 378.731,A -85,B 0,C 180,E1 -6341.781,E2 -6341.781} C_VEL
LIN {X 0,Y 495.74,Z 378.733,A -85,B 0,C 180,E1 -6345.141,E2 -6345.141} C_VEL
LIN {X 0,Y 495.781,Z 378.727,A -85,B 0,C 180,E1 -6348.221,E2 -6348.221} C_VEL
LIN {X 0,Y 495.753,Z 378.735,A -85,B 0,C 180,E1 -6351.408,E2 -6351.408} C_VEL
LIN {X 0,Y 495.668,Z 378.743,A -85,B 0,C 180,E1 -6354.456,E2 -6354.456} C_VEL
LIN {X 0,Y 495.389,Z 378.836,A -85,B 0,C 180,E1 -6357.377,E2 -6357.377} C_VEL
LIN {X 0,Y 495.358,Z 381.669,A -85,B 0,C 180,E1 -6360.227,E2 -6360.227} C_VEL
LIN {X 0,Y 495.322,Z 382.165,A -85,B 0,C 180,E1 -6360.719,E2 -6360.719} C_VEL
LIN {X 0,Y 494.635,Z 382.912,A -85,B 0,C 180,E1 -6361.392,E2 -6361.392} C_VEL
LIN {X 0,Y 491.74,Z 384.299,A -85,B 0,C 180,E1 -6362.482,E2 -6362.482} C_VEL
LIN {X 0,Y 489.305,Z 385.419,A -85,B 0,C 180,E1 -6363.36,E2 -6363.36} C_VEL
LIN {X 0,Y 488.268,Z 386.199,A -85,B 0,C 180,E1 -6364.04,E2 -6364.04} C_VEL
LIN {X 0,Y 488.189,Z 386.437,A -85,B 0,C 180,E1 -6364.271,E2 -6364.271} C_VEL
LIN {X 0,Y 488.147,Z 389.354,A -85,B 0,C 180,E1 -6367.136,E2 -6367.136} C_VEL
LIN {X 0,Y 488.086,Z 392.132,A -85,B 0,C 180,E1 -6369.783,E2 -6369.783} C_VEL
LIN {X 0,Y 488.064,Z 395.031,A -85,B 0,C 180,E1 -6372.398,E2 -6372.398} C_VEL
LIN {X 0,Y 488.07,Z 398.538,A -85,B 0,C 180,E1 -6375.378,E2 -6375.378} C_VEL
LIN {X 0,Y 490.795,Z 411.078,A -85,B 0,C 180,E1 -6375.818,E2 -6375.818} C_VEL
LIN {X 0,Y 490.734,Z 423.494,A -85,B 0,C 180,E1 -6376.332,E2 -6376.332} C_VEL
LIN {X 0,Y 490.391,Z 435.187,A -85,B 0,C 180,E1 -6376.976,E2 -6376.976} C_VEL
LIN {X 0,Y 489.975,Z 446.492,A -85,B 0,C 180,E1 -6377.786,E2 -6377.786} C_VEL
LIN {X 0,Y 489.587,Z 456.923,A -85,B 0,C 180,E1 -6378.721,E2 -6378.721} C_VEL
LIN {X 0,Y 489.21,Z 465.444,A -85,B 0,C 180,E1 -6379.655,E2 -6379.655} C_VEL
LIN {X 0,Y 488.907,Z 473.283,A -85,B 0,C 180,E1 -6380.693,E2 -6380.693} C_VEL
LIN {X 0,Y 488.555,Z 480.949,A -85,B 0,C 180,E1 -6381.937,E2 -6381.937} C_VEL
LIN {X 0,Y 488.31,Z 487.971,A -85,B 0,C 180,E1 -6383.388,E2 -6383.388} C_VEL
LIN {X 0,Y 488.079,Z 492.654,A -85,B 0,C 180,E1 -6384.63,E2 -6384.63} C_VEL
LIN {X 0,Y 488.11,Z 496.227,A -85,B 0,C 180,E1 -6385.872,E2 -6385.872} C_VEL
LIN {X 0,Y 488.059,Z 498.078,A -85,B 0,C 180,E1 -6386.698,E2 -6386.698} C_VEL
LIN {X 0,Y 487.999,Z 499.475,A -85,B 0,C 180,E1 -6387.524,E2 -6387.524} C_VEL
LIN {X 0,Y 487.838,Z 501.085,A -85,B 0,C 180,E1 -6389.175,E2 -6389.175} C_VEL
LIN {X 0,Y 487.827,Z 501.32,A -85,B 0,C 180,E1 -6390,E2 -6390} C_VEL
LIN {X 0,Y 487.838,Z 501.136,A -85,B 0,C 180,E1 -6390.826,E2 -6390.826} C_VEL
LIN {X 0,Y 488,Z 499.592,A -85,B 0,C 180,E1 -6392.476,E2 -6392.476} C_VEL
LIN {X 0,Y 488.059,Z 498.246,A -85,B 0,C 180,E1 -6393.302,E2 -6393.302} C_VEL
LIN {X 0,Y 488.089,Z 495.406,A -85,B 0,C 180,E1 -6394.542,E2 -6394.542} C_VEL
LIN {X 0,Y 488.191,Z 491.55,A -85,B 0,C 180,E1 -6395.784,E2 -6395.784} C_VEL
LIN {X 0,Y 488.329,Z 486.575,A -85,B 0,C 180,E1 -6397.026,E2 -6397.026} C_VEL
LIN {X 0,Y 488.616,Z 480.302,A -85,B 0,C 180,E1 -6398.27,E2 -6398.27} C_VEL
LIN {X 0,Y 488.879,Z 472.45,A -85,B 0,C 180,E1 -6399.516,E2 -6399.516} C_VEL
LIN {X 0,Y 489.364,Z 462.668,A -85,B 0,C 180,E1 -6400.76,E2 -6400.76} C_VEL
LIN {X 0,Y 489.785,Z 452.403,A -85,B 0,C 180,E1 -6401.799,E2 -6401.799} C_VEL
LIN {X 0,Y 490.168,Z 442.101,A -85,B 0,C 180,E1 -6402.64,E2 -6402.64} C_VEL
LIN {X 0,Y 490.487,Z 431.094,A -85,B 0,C 180,E1 -6403.359,E2 -6403.359} C_VEL
LIN {X 0,Y 490.839,Z 418.565,A -85,B 0,C 180,E1 -6403.982,E2 -6403.982} C_VEL
LIN {X 0,Y 490.723,Z 410.634,A -85,B 0,C 180,E1 -6404.29,E2 -6404.29} C_VEL
LIN {X 0,Y 488.053,Z 398.476,A -85,B 0,C 180,E1 -6404.729,E2 -6404.729} C_VEL
LIN {X 0,Y 488.057,Z 394.552,A -85,B 0,C 180,E1 -6408.121,E2 -6408.121} C_VEL
LIN {X 0,Y 488.073,Z 391.278,A -85,B 0,C 180,E1 -6411.1,E2 -6411.1} C_VEL
LIN {X 0,Y 488.114,Z 388.497,A -85,B 0,C 180,E1 -6413.776,E2 -6413.776} C_VEL
LIN {X 0,Y 488.222,Z 385.712,A -85,B 0,C 180,E1 -6416.503,E2 -6416.503} C_VEL
LIN {X 0,Y 488.271,Z 382.933,A -85,B 0,C 180,E1 -6419.3,E2 -6419.3} C_VEL
LIN {X 0,Y 488.325,Z 380.099,A -85,B 0,C 180,E1 -6422.175,E2 -6422.175} C_VEL
LIN {X 0,Y 488.445,Z 379.643,A -85,B 0,C 180,E1 -6423.432,E2 -6423.432} C_VEL
LIN {X 0,Y 488.661,Z 379.615,A -85,B 0,C 180,E1 -6426.351,E2 -6426.351} C_VEL
LIN {X 0,Y 488.705,Z 379.608,A -85,B 0,C 180,E1 -6429.254,E2 -6429.254} C_VEL
LIN {X 0,Y 488.712,Z 379.606,A -85,B 0,C 180,E1 -6431.6,E2 -6431.6} C_VEL
LIN {X 0,Y 488.705,Z 379.609,A -85,B 0,C 180,E1 -6434.803,E2 -6434.803} C_VEL
LIN {X 0,Y 488.696,Z 379.612,A -85,B 0,C 180,E1 -6437.475,E2 -6437.475} C_VEL
LIN {X 0,Y 488.737,Z 379.606,A -85,B 0,C 180,E1 -6439.677,E2 -6439.677} C_VEL
LIN {X 0,Y 488.687,Z 379.611,A -85,B 0,C 180,E1 -6442.842,E2 -6442.842} C_VEL
LIN {X 0,Y 488.739,Z 379.608,A -85,B 0,C 180,E1 -6445.888,E2 -6445.888} C_VEL
LIN {X 0,Y 488.697,Z 379.611,A -85,B 0,C 180,E1 -6448.82,E2 -6448.82} C_VEL
LIN {X 0,Y 488.749,Z 379.604,A -85,B 0,C 180,E1 -6451.671,E2 -6451.671} C_VEL
LIN {X 0,Y 488.732,Z 379.609,A -85,B 0,C 180,E1 -6454.443,E2 -6454.443} C_VEL
LIN {X 0,Y 488.727,Z 379.604,A -85,B 0,C 180,E1 -6457.153,E2 -6457.153} C_VEL
LIN {X 0,Y 488.734,Z 379.609,A -85,B 0,C 180,E1 -6459.811,E2 -6459.811} C_VEL
LIN {X 0,Y 488.72,Z 379.608,A -85,B 0,C 180,E1 -6462.423,E2 -6462.423} C_VEL
LIN {X 0,Y 488.767,Z 379.602,A -85,B 0,C 180,E1 -6465,E2 -6465} C_VEL
LIN {X 0,Y 488.811,Z 379.596,A -85,B 0,C 180,E1 -6468.388,E2 -6468.388} C_VEL
LIN {X 0,Y 488.791,Z 379.602,A -85,B 0,C 180,E1 -6471.733,E2 -6471.733} C_VEL
LIN {X 0,Y 488.86,Z 379.59,A -85,B 0,C 180,E1 -6474.224,E2 -6474.224} C_VEL
LIN {X 0,Y 488.964,Z 379.577,A -85,B 0,C 180,E1 -6477.529,E2 -6477.529} C_VEL
LIN {X 0,Y 488.94,Z 379.579,A -85,B 0,C 180,E1 -6480.824,E2 -6480.824} C_VEL
LIN {X 0,Y 488.966,Z 379.574,A -85,B 0,C 180,E1 -6482.471,E2 -6482.471} C_VEL
LIN {X 0,Y 488.86,Z 379.59,A -85,B 0,C 180,E1 -6485.776,E2 -6485.776} C_VEL
LIN {X 0,Y 488.823,Z 379.596,A -85,B 0,C 180,E1 -6488.266,E2 -6488.266} C_VEL
LIN {X 0,Y 488.835,Z 379.594,A -85,B 0,C 180,E1 -6491.612,E2 -6491.612} C_VEL
LIN {X 0,Y 488.767,Z 379.601,A -85,B 0,C 180,E1 -6495,E2 -6495} C_VEL
LIN {X 0,Y 488.752,Z 379.603,A -85,B 0,C 180,E1 -6498.442,E2 -6498.442} C_VEL
LIN {X 0,Y 488.712,Z 379.61,A -85,B 0,C 180,E1 -6501.071,E2 -6501.071} C_VEL
LIN {X 0,Y 488.685,Z 379.615,A -85,B 0,C 180,E1 -6503.746,E2 -6503.746} C_VEL
LIN {X 0,Y 488.797,Z 379.598,A -85,B 0,C 180,E1 -6506.944,E2 -6506.944} C_VEL
LIN {X 0,Y 488.714,Z 379.607,A -85,B 0,C 180,E1 -6510.363,E2 -6510.363} C_VEL
LIN {X 0,Y 488.739,Z 379.605,A -85,B 0,C 180,E1 -6513.484,E2 -6513.484} C_VEL
LIN {X 0,Y 488.686,Z 379.613,A -85,B 0,C 180,E1 -6516.354,E2 -6516.354} C_VEL
LIN {X 0,Y 488.706,Z 379.613,A -85,B 0,C 180,E1 -6519.254,E2 -6519.254} C_VEL
LIN {X 0,Y 488.711,Z 379.611,A -85,B 0,C 180,E1 -6521.6,E2 -6521.6} C_VEL
LIN {X 0,Y 488.716,Z 379.611,A -85,B 0,C 180,E1 -6524.801,E2 -6524.801} C_VEL
LIN {X 0,Y 488.699,Z 379.613,A -85,B 0,C 180,E1 -6527.475,E2 -6527.475} C_VEL
LIN {X 0,Y 488.743,Z 379.668,A -85,B 0,C 180,E1 -6530.349,E2 -6530.349} C_VEL
LIN {X 0,Y 490.046,Z 387.075,A -85,B 0,C 180,E1 -6533.43,E2 -6533.43} C_VEL
LIN {X 0,Y 490.183,Z 391.222,A -85,B 0,C 180,E1 -6535.005,E2 -6535.005} C_VEL
LIN {X 0,Y 489.902,Z 399.34,A -85,B 0,C 180,E1 -6537.941,E2 -6537.941} C_VEL
LIN {X 0,Y 489.564,Z 408.491,A -85,B 0,C 180,E1 -6541.128,E2 -6541.128} C_VEL
LIN {X 0,Y 489.306,Z 415.636,A -85,B 0,C 180,E1 -6543.56,E2 -6543.56} C_VEL
LIN {X 0,Y 489.062,Z 423.83,A -85,B 0,C 180,E1 -6546.273,E2 -6546.273} C_VEL
LIN {X 0,Y 488.83,Z 433.743,A -85,B 0,C 180,E1 -6549.48,E2 -6549.48} C_VEL
LIN {X 0,Y 488.583,Z 442.759,A -85,B 0,C 180,E1 -6552.418,E2 -6552.418} C_VEL
LIN {X 0,Y 488.388,Z 451.581,A -85,B 0,C 180,E1 -6555.271,E2 -6555.271} C_VEL
LIN {X 0,Y 490.683,Z 465.089,A -85,B 0,C 180,E1 -6555.669,E2 -6555.669} C_VEL
LIN {X 0,Y 490.769,Z 471.869,A -85,B 0,C 180,E1 -6555.91,E2 -6555.91} C_VEL
LIN {X 0,Y 490.402,Z 483.5,A -85,B 0,C 180,E1 -6556.428,E2 -6556.428} C_VEL
LIN {X 0,Y 490,Z 495.31,A -85,B 0,C 180,E1 -6557.123,E2 -6557.123} C_VEL
LIN {X 0,Y 489.656,Z 506.742,A -85,B 0,C 180,E1 -6557.988,E2 -6557.988} C_VEL
LIN {X 0,Y 489.283,Z 515.645,A -85,B 0,C 180,E1 -6558.819,E2 -6558.819} C_VEL
LIN {X 0,Y 488.893,Z 524.784,A -85,B 0,C 180,E1 -6559.857,E2 -6559.857} C_VEL
LIN {X 0,Y 488.578,Z 533.687,A -85,B 0,C 180,E1 -6561.104,E2 -6561.104} C_VEL
LIN {X 0,Y 488.251,Z 540.848,A -85,B 0,C 180,E1 -6562.348,E2 -6562.348} C_VEL
LIN {X 0,Y 488.096,Z 547.062,A -85,B 0,C 180,E1 -6563.722,E2 -6563.722} C_VEL
LIN {X 0,Y 487.971,Z 551.676,A -85,B 0,C 180,E1 -6565.042,E2 -6565.042} C_VEL
LIN {X 0,Y 487.947,Z 553.958,A -85,B 0,C 180,E1 -6565.87,E2 -6565.87} C_VEL
LIN {X 0,Y 487.966,Z 555.807,A -85,B 0,C 180,E1 -6566.697,E2 -6566.697} C_VEL
LIN {X 0,Y 487.889,Z 558.183,A -85,B 0,C 180,E1 -6568.349,E2 -6568.349} C_VEL
LIN {X 0,Y 487.819,Z 559,A -85,B 0,C 180,E1 -6570,E2 -6570} C_VEL
LIN {X 0,Y 487.889,Z 558.184,A -85,B 0,C 180,E1 -6571.651,E2 -6571.651} C_VEL
LIN {X 0,Y 487.966,Z 555.81,A -85,B 0,C 180,E1 -6573.303,E2 -6573.303} C_VEL
LIN {X 0,Y 487.938,Z 552.895,A -85,B 0,C 180,E1 -6574.544,E2 -6574.544} C_VEL
LIN {X 0,Y 488.104,Z 548.948,A -85,B 0,C 180,E1 -6575.785,E2 -6575.785} C_VEL
LIN {X 0,Y 488.19,Z 542.876,A -85,B 0,C 180,E1 -6577.236,E2 -6577.236} C_VEL
LIN {X 0,Y 488.454,Z 536.236,A -85,B 0,C 180,E1 -6578.481,E2 -6578.481} C_VEL
LIN {X 0,Y 488.761,Z 527.992,A -85,B 0,C 180,E1 -6579.727,E2 -6579.727} C_VEL
LIN {X 0,Y 489.081,Z 519.54,A -85,B 0,C 180,E1 -6580.767,E2 -6580.767} C_VEL
LIN {X 0,Y 489.575,Z 509.092,A -85,B 0,C 180,E1 -6581.804,E2 -6581.804} C_VEL
LIN {X 0,Y 489.931,Z 497.602,A -85,B 0,C 180,E1 -6582.721,E2 -6582.721} C_VEL
LIN {X 0,Y 490.369,Z 485.487,A -85,B 0,C 180,E1 -6583.468,E2 -6583.468} C_VEL
LIN {X 0,Y 490.755,Z 473.165,A -85,B 0,C 180,E1 -6584.038,E2 -6584.038} C_VEL
LIN {X 0,Y 490.651,Z 465.086,A -85,B 0,C 180,E1 -6584.332,E2 -6584.332} C_VEL
LIN {X 0,Y 488.396,Z 451.53,A -85,B 0,C 180,E1 -6584.745,E2 -6584.745} C_VEL
LIN {X 0,Y 488.621,Z 441.612,A -85,B 0,C 180,E1 -6587.956,E2 -6587.956} C_VEL
LIN {X 0,Y 488.862,Z 432.036,A -85,B 0,C 180,E1 -6591.064,E2 -6591.064} C_VEL
LIN {X 0,Y 489.094,Z 422.429,A -85,B 0,C 180,E1 -6594.175,E2 -6594.175} C_VEL
LIN {X 0,Y 489.459,Z 412.909,A -85,B 0,C 180,E1 -6597.354,E2 -6597.354} C_VEL
LIN {X 0,Y 489.744,Z 403.557,A -85,B 0,C 180,E1 -6600.568,E2 -6600.568} C_VEL
LIN {X 0,Y 490.09,Z 394.698,A -85,B 0,C 180,E1 -6603.723,E2 -6603.723} C_VEL
LIN {X 0,Y 490.227,Z 388.536,A -85,B 0,C 180,E1 -6606,E2 -6606} C_VEL
LIN {X 0,Y 489.17,Z 382.094,A -85,B 0,C 180,E1 -6608.613,E2 -6608.613} C_VEL
LIN {X 0,Y 488.715,Z 379.612,A -85,B 0,C 180,E1 -6609.72,E2 -6609.72} C_VEL
LIN {X 0,Y 488.718,Z 379.612,A -85,B 0,C 180,E1 -6612.827,E2 -6612.827} C_VEL
LIN {X 0,Y 488.702,Z 379.61,A -85,B 0,C 180,E1 -6615.976,E2 -6615.976} C_VEL
LIN {X 0,Y 488.711,Z 379.609,A -85,B 0,C 180,E1 -6618.585,E2 -6618.585} C_VEL
LIN {X 0,Y 488.708,Z 379.61,A -85,B 0,C 180,E1 -6620.947,E2 -6620.947} C_VEL
LIN {X 0,Y 488.686,Z 379.613,A -85,B 0,C 180,E1 -6623.869,E2 -6623.869} C_VEL
LIN {X 0,Y 488.742,Z 379.606,A -85,B 0,C 180,E1 -6626.877,E2 -6626.877} C_VEL
LIN {X 0,Y 488.727,Z 379.605,A -85,B 0,C 180,E1 -6629.781,E2 -6629.781} C_VEL
LIN {X 0,Y 488.795,Z 379.598,A -85,B 0,C 180,E1 -6633.056,E2 -6633.056} C_VEL
LIN {X 0,Y 488.684,Z 379.615,A -85,B 0,C 180,E1 -6636.254,E2 -6636.254} C_VEL
LIN {X 0,Y 488.75,Z 379.607,A -85,B 0,C 180,E1 -6639.176,E2 -6639.176} C_VEL
LIN {X 0,Y 488.763,Z 379.602,A -85,B 0,C 180,E1 -6641.628,E2 -6641.628} C_VEL
LIN {X 0,Y 488.766,Z 379.601,A -85,B 0,C 180,E1 -6645,E2 -6645} C_VEL
LIN {X 0,Y 488.834,Z 379.595,A -85,B 0,C 180,E1 -6648.388,E2 -6648.388} C_VEL
LIN {X 0,Y 488.822,Z 379.596,A -85,B 0,C 180,E1 -6651.734,E2 -6651.734} C_VEL
LIN {X 0,Y 488.858,Z 379.59,A -85,B 0,C 180,E1 -6654.224,E2 -6654.224} C_VEL
LIN {X 0,Y 488.965,Z 379.574,A -85,B 0,C 180,E1 -6657.529,E2 -6657.529} C_VEL
LIN {X 0,Y 488.958,Z 379.577,A -85,B 0,C 180,E1 -6660.824,E2 -6660.824} C_VEL
LIN {X 0,Y 488.963,Z 379.577,A -85,B 0,C 180,E1 -6662.471,E2 -6662.471} C_VEL
LIN {X 0,Y 488.859,Z 379.59,A -85,B 0,C 180,E1 -6665.776,E2 -6665.776} C_VEL
LIN {X 0,Y 488.819,Z 379.598,A -85,B 0,C 180,E1 -6668.266,E2 -6668.266} C_VEL
LIN {X 0,Y 488.81,Z 379.596,A -85,B 0,C 180,E1 -6671.612,E2 -6671.612} C_VEL
LIN {X 0,Y 488.766,Z 379.603,A -85,B 0,C 180,E1 -6675,E2 -6675} C_VEL
LIN {X 0,Y 488.751,Z 379.606,A -85,B 0,C 180,E1 -6678.442,E2 -6678.442} C_VEL
LIN {X 0,Y 488.711,Z 379.608,A -85,B 0,C 180,E1 -6681.071,E2 -6681.071} C_VEL
LIN {X 0,Y 488.684,Z 379.614,A -85,B 0,C 180,E1 -6683.746,E2 -6683.746} C_VEL
LIN {X 0,Y 488.796,Z 379.598,A -85,B 0,C 180,E1 -6686.944,E2 -6686.944} C_VEL
LIN {X 0,Y 488.713,Z 379.611,A -85,B 0,C 180,E1 -6690.363,E2 -6690.363} C_VEL
LIN {X 0,Y 488.738,Z 379.605,A -85,B 0,C 180,E1 -6693.484,E2 -6693.484} C_VEL
LIN {X 0,Y 488.686,Z 379.61,A -85,B 0,C 180,E1 -6696.355,E2 -6696.355} C_VEL
LIN {X 0,Y 488.705,Z 379.611,A -85,B 0,C 180,E1 -6699.254,E2 -6699.254} C_VEL
LIN {X 0,Y 488.711,Z 379.609,A -85,B 0,C 180,E1 -6701.6,E2 -6701.6} C_VEL
LIN {X 0,Y 488.704,Z 379.61,A -85,B 0,C 180,E1 -6704.803,E2 -6704.803} C_VEL
LIN {X 0,Y 488.739,Z 379.606,A -85,B 0,C 180,E1 -6707.479,E2 -6707.479} C_VEL
LIN {X 0,Y 488.704,Z 379.608,A -85,B 0,C 180,E1 -6710.746,E2 -6710.746} C_VEL
LIN {X 0,Y 488.652,Z 379.616,A -85,B 0,C 180,E1 -6713.866,E2 -6713.866} C_VEL
LIN {X 0,Y 488.423,Z 379.649,A -85,B 0,C 180,E1 -6716.853,E2 -6716.853} C_VEL
LIN {X 0,Y 488.338,Z 380.291,A -85,B 0,C 180,E1 -6718.115,E2 -6718.115} C_VEL
LIN {X 0,Y 488.292,Z 383.55,A -85,B 0,C 180,E1 -6721.4,E2 -6721.4} C_VEL
LIN {X 0,Y 488.189,Z 386.437,A -85,B 0,C 180,E1 -6724.271,E2 -6724.271} C_VEL
LIN {X 0,Y 487.528,Z 387.199,A -85,B 0,C 180,E1 -6724.954,E2 -6724.954} C_VEL
LIN {X 0,Y 484.646,Z 388.595,A -85,B 0,C 180,E1 -6726.059,E2 -6726.059} C_VEL
LIN {X 0,Y 482.188,Z 389.73,A -85,B 0,C 180,E1 -6726.949,E2 -6726.949} C_VEL
LIN {X 0,Y 481.115,Z 390.531,A -85,B 0,C 180,E1 -6727.639,E2 -6727.639} C_VEL
LIN {X 0,Y 481.019,Z 390.778,A -85,B 0,C 180,E1 -6727.873,E2 -6727.873} C_VEL
LIN {X 0,Y 480.998,Z 393.423,A -85,B 0,C 180,E1 -6730.363,E2 -6730.363} C_VEL
LIN {X 0,Y 480.964,Z 396.374,A -85,B 0,C 180,E1 -6733.007,E2 -6733.007} C_VEL
LIN {X 0,Y 481.007,Z 399.004,A -85,B 0,C 180,E1 -6735.158,E2 -6735.158} C_VEL
LIN {X 0,Y 483.952,Z 412.283,A -85,B 0,C 180,E1 -6735.64,E2 -6735.64} C_VEL
LIN {X 0,Y 483.829,Z 425.046,A -85,B 0,C 180,E1 -6736.186,E2 -6736.186} C_VEL
LIN {X 0,Y 483.449,Z 437.383,A -85,B 0,C 180,E1 -6736.905,E2 -6736.905} C_VEL
LIN {X 0,Y 483.014,Z 448.213,A -85,B 0,C 180,E1 -6737.714,E2 -6737.714} C_VEL
LIN {X 0,Y 482.612,Z 458.417,A -85,B 0,C 180,E1 -6738.662,E2 -6738.662} C_VEL
LIN {X 0,Y 482.171,Z 467.572,A -85,B 0,C 180,E1 -6739.715,E2 -6739.715} C_VEL
LIN {X 0,Y 481.798,Z 476.446,A -85,B 0,C 180,E1 -6740.978,E2 -6740.978} C_VEL
LIN {X 0,Y 481.455,Z 483.59,A -85,B 0,C 180,E1 -6742.24,E2 -6742.24} C_VEL
LIN {X 0,Y 481.253,Z 489.416,A -85,B 0,C 180,E1 -6743.534,E2 -6743.534} C_VEL
LIN {X 0,Y 480.959,Z 494.397,A -85,B 0,C 180,E1 -6744.97,E2 -6744.97} C_VEL
LIN {X 0,Y 481.05,Z 496.66,A -85,B 0,C 180,E1 -6745.811,E2 -6745.811} C_VEL
LIN {X 0,Y 480.984,Z 498.511,A -85,B 0,C 180,E1 -6746.649,E2 -6746.649} C_VEL
LIN {X 0,Y 480.939,Z 499.906,A -85,B 0,C 180,E1 -6747.487,E2 -6747.487} C_VEL
LIN {X 0,Y 480.764,Z 501.516,A -85,B 0,C 180,E1 -6749.162,E2 -6749.162} C_VEL
LIN {X 0,Y 480.75,Z 501.751,A -85,B 0,C 180,E1 -6750,E2 -6750} C_VEL
LIN {X 0,Y 480.764,Z 501.567,A -85,B 0,C 180,E1 -6750.838,E2 -6750.838} C_VEL
LIN {X 0,Y 480.94,Z 500.021,A -85,B 0,C 180,E1 -6752.513,E2 -6752.513} C_VEL
LIN {X 0,Y 480.984,Z 498.677,A -85,B 0,C 180,E1 -6753.351,E2 -6753.351} C_VEL
LIN {X 0,Y 481.026,Z 495.836,A -85,B 0,C 180,E1 -6754.609,E2 -6754.609} C_VEL
LIN {X 0,Y 481.145,Z 491.979,A -85,B 0,C 180,E1 -6755.869,E2 -6755.869} C_VEL
LIN {X 0,Y 481.287,Z 487.005,A -85,B 0,C 180,E1 -6757.13,E2 -6757.13} C_VEL
LIN {X 0,Y 481.594,Z 480.73,A -85,B 0,C 180,E1 -6758.391,E2 -6758.391} C_VEL
LIN {X 0,Y 481.883,Z 472.878,A -85,B 0,C 180,E1 -6759.656,E2 -6759.656} C_VEL
LIN {X 0,Y 482.392,Z 463.094,A -85,B 0,C 180,E1 -6760.918,E2 -6760.918} C_VEL
LIN {X 0,Y 482.853,Z 452.827,A -85,B 0,C 180,E1 -6761.971,E2 -6761.971} C_VEL
LIN {X 0,Y 483.248,Z 442.842,A -85,B 0,C 180,E1 -6762.8,E2 -6762.8} C_VEL
LIN {X 0,Y 483.618,Z 431.514,A -85,B 0,C 180,E1 -6763.552,E2 -6763.552} C_VEL
LIN {X 0,Y 483.981,Z 418.981,A -85,B 0,C 180,E1 -6764.185,E2 -6764.185} C_VEL
LIN {X 0,Y 483.885,Z 411.806,A -85,B 0,C 180,E1 -6764.469,E2 -6764.469} C_VEL
LIN {X 0,Y 480.986,Z 398.866,A -85,B 0,C 180,E1 -6764.951,E2 -6764.951} C_VEL
LIN {X 0,Y 480.98,Z 395.079,A -85,B 0,C 180,E1 -6768.236,E2 -6768.236} C_VEL
LIN {X 0,Y 481.001,Z 391.6,A -85,B 0,C 180,E1 -6771.425,E2 -6771.425} C_VEL
LIN {X 0,Y 481.082,Z 388.8,A -85,B 0,C 180,E1 -6774.145,E2 -6774.145} C_VEL
LIN {X 0,Y 481.172,Z 385.904,A -85,B 0,C 180,E1 -6777.005,E2 -6777.005} C_VEL
LIN {X 0,Y 481.221,Z 383.178,A -85,B 0,C 180,E1 -6779.773,E2 -6779.773} C_VEL
LIN {X 0,Y 481.283,Z 380.881,A -85,B 0,C 180,E1 -6782.118,E2 -6782.118} C_VEL
LIN {X 0,Y 481.304,Z 380.534,A -85,B 0,C 180,E1 -6782.703,E2 -6782.703} C_VEL
LIN {X 0,Y 481.585,Z 380.497,A -85,B 0,C 180,E1 -6785.714,E2 -6785.714} C_VEL
LIN {X 0,Y 481.674,Z 380.487,A -85,B 0,C 180,E1 -6788.859,E2 -6788.859} C_VEL
LIN {X 0,Y 481.657,Z 380.487,A -85,B 0,C 180,E1 -6791.913,E2 -6791.913} C_VEL
LIN {X 0,Y 481.659,Z 380.488,A -85,B 0,C 180,E1 -6794.458,E2 -6794.458} C_VEL
LIN {X 0,Y 481.651,Z 380.49,A -85,B 0,C 180,E1 -6797.839,E2 -6797.839} C_VEL
LIN {X 0,Y 481.685,Z 380.487,A -85,B 0,C 180,E1 -6800.651,E2 -6800.651} C_VEL
LIN {X 0,Y 481.635,Z 380.487,A -85,B 0,C 180,E1 -6803.376,E2 -6803.376} C_VEL
LIN {X 0,Y 481.714,Z 380.481,A -85,B 0,C 180,E1 -6806.33,E2 -6806.33} C_VEL
LIN {X 0,Y 481.655,Z 380.489,A -85,B 0,C 180,E1 -6809.417,E2 -6809.417} C_VEL
LIN {X 0,Y 481.705,Z 380.482,A -85,B 0,C 180,E1 -6812.168,E2 -6812.168} C_VEL
LIN {X 0,Y 481.698,Z 380.481,A -85,B 0,C 180,E1 -6814.969,E2 -6814.969} C_VEL
LIN {X 0,Y 481.654,Z 380.489,A -85,B 0,C 180,E1 -6817.705,E2 -6817.705} C_VEL
LIN {X 0,Y 481.713,Z 380.48,A -85,B 0,C 180,E1 -6820.393,E2 -6820.393} C_VEL
LIN {X 0,Y 481.685,Z 380.485,A -85,B 0,C 180,E1 -6823.034,E2 -6823.034} C_VEL
LIN {X 0,Y 481.695,Z 380.483,A -85,B 0,C 180,E1 -6825.639,E2 -6825.639} C_VEL
LIN {X 0,Y 481.756,Z 380.477,A -85,B 0,C 180,E1 -6828.215,E2 -6828.215} C_VEL
LIN {X 0,Y 481.745,Z 380.48,A -85,B 0,C 180,E1 -6831.611,E2 -6831.611} C_VEL
LIN {X 0,Y 481.821,Z 380.467,A -85,B 0,C 180,E1 -6834.14,E2 -6834.14} C_VEL
LIN {X 0,Y 481.931,Z 380.453,A -85,B 0,C 180,E1 -6837.493,E2 -6837.493} C_VEL
LIN {X 0,Y 481.892,Z 380.457,A -85,B 0,C 180,E1 -6840.836,E2 -6840.836} C_VEL
LIN {X 0,Y 481.933,Z 380.45,A -85,B 0,C 180,E1 -6842.507,E2 -6842.507} C_VEL
LIN {X 0,Y 481.821,Z 380.467,A -85,B 0,C 180,E1 -6845.86,E2 -6845.86} C_VEL
LIN {X 0,Y 481.769,Z 380.474,A -85,B 0,C 180,E1 -6848.388,E2 -6848.388} C_VEL
LIN {X 0,Y 481.8,Z 380.472,A -85,B 0,C 180,E1 -6851.784,E2 -6851.784} C_VEL
LIN {X 0,Y 481.748,Z 380.477,A -85,B 0,C 180,E1 -6855.224,E2 -6855.224} C_VEL
LIN {X 0,Y 481.714,Z 380.48,A -85,B 0,C 180,E1 -6858.722,E2 -6858.722} C_VEL
LIN {X 0,Y 481.65,Z 380.489,A -85,B 0,C 180,E1 -6861.395,E2 -6861.395} C_VEL
LIN {X 0,Y 481.666,Z 380.487,A -85,B 0,C 180,E1 -6864.114,E2 -6864.114} C_VEL
LIN {X 0,Y 481.752,Z 380.477,A -85,B 0,C 180,E1 -6867.139,E2 -6867.139} C_VEL
LIN {X 0,Y 481.683,Z 380.483,A -85,B 0,C 180,E1 -6869.741,E2 -6869.741} C_VEL
LIN {X 0,Y 481.676,Z 380.487,A -85,B 0,C 180,E1 -6872.674,E2 -6872.674} C_VEL
LIN {X 0,Y 481.641,Z 380.492,A -85,B 0,C 180,E1 -6875.709,E2 -6875.709} C_VEL
LIN {X 0,Y 481.675,Z 380.485,A -85,B 0,C 180,E1 -6878.859,E2 -6878.859} C_VEL
LIN {X 0,Y 481.656,Z 380.489,A -85,B 0,C 180,E1 -6881.913,E2 -6881.913} C_VEL
LIN {X 0,Y 481.663,Z 380.489,A -85,B 0,C 180,E1 -6884.457,E2 -6884.457} C_VEL
LIN {X 0,Y 481.658,Z 380.491,A -85,B 0,C 180,E1 -6887.84,E2 -6887.84} C_VEL
LIN {X 0,Y 481.702,Z 380.538,A -85,B 0,C 180,E1 -6890.062,E2 -6890.062} C_VEL
LIN {X 0,Y 482.985,Z 387.844,A -85,B 0,C 180,E1 -6893.16,E2 -6893.16} C_VEL
LIN {X 0,Y 483.253,Z 391.33,A -85,B 0,C 180,E1 -6894.53,E2 -6894.53} C_VEL
LIN {X 0,Y 482.959,Z 399.14,A -85,B 0,C 180,E1 -6897.423,E2 -6897.423} C_VEL
LIN {X 0,Y 482.603,Z 407.278,A -85,B 0,C 180,E1 -6900.321,E2 -6900.321} C_VEL
LIN {X 0,Y 482.332,Z 415.41,A -85,B 0,C 180,E1 -6903.147,E2 -6903.147} C_VEL
LIN {X 0,Y 482.003,Z 424.93,A -85,B 0,C 180,E1 -6906.361,E2 -6906.361} C_VEL
LIN {X 0,Y 481.773,Z 434.5,A -85,B 0,C 180,E1 -6909.506,E2 -6909.506} C_VEL
LIN {X 0,Y 481.505,Z 444.076,A -85,B 0,C 180,E1 -6912.589,E2 -6912.589} C_VEL
LIN {X 0,Y 481.342,Z 451.718,A -85,B 0,C 180,E1 -6915.054,E2 -6915.054} C_VEL
LIN {X 0,Y 483.671,Z 465.089,A -85,B 0,C 180,E1 -6915.457,E2 -6915.457} C_VEL
LIN {X 0,Y 483.968,Z 469.735,A -85,B 0,C 180,E1 -6915.627,E2 -6915.627} C_VEL
LIN {X 0,Y 483.572,Z 482.507,A -85,B 0,C 180,E1 -6916.179,E2 -6916.179} C_VEL
LIN {X 0,Y 483.136,Z 494.202,A -85,B 0,C 180,E1 -6916.862,E2 -6916.862} C_VEL
LIN {X 0,Y 482.762,Z 505.483,A -85,B 0,C 180,E1 -6917.707,E2 -6917.707} C_VEL
LIN {X 0,Y 482.326,Z 515.644,A -85,B 0,C 180,E1 -6918.655,E2 -6918.655} C_VEL
LIN {X 0,Y 481.878,Z 524.784,A -85,B 0,C 180,E1 -6919.708,E2 -6919.708} C_VEL
LIN {X 0,Y 481.531,Z 533.687,A -85,B 0,C 180,E1 -6920.973,E2 -6920.973} C_VEL
LIN {X 0,Y 481.208,Z 540.848,A -85,B 0,C 180,E1 -6922.236,E2 -6922.236} C_VEL
LIN {X 0,Y 481.048,Z 546.357,A -85,B 0,C 180,E1 -6923.447,E2 -6923.447} C_VEL
LIN {X 0,Y 480.998,Z 550.372,A -85,B 0,C 180,E1 -6924.55,E2 -6924.55} C_VEL
LIN {X 0,Y 480.847,Z 553.958,A -85,B 0,C 180,E1 -6925.809,E2 -6925.809} C_VEL
LIN {X 0,Y 480.891,Z 555.807,A -85,B 0,C 180,E1 -6926.649,E2 -6926.649} C_VEL
LIN {X 0,Y 480.79,Z 558.182,A -85,B 0,C 180,E1 -6928.325,E2 -6928.325} C_VEL
LIN {X 0,Y 480.743,Z 559,A -85,B 0,C 180,E1 -6930,E2 -6930} C_VEL
LIN {X 0,Y 480.79,Z 558.184,A -85,B 0,C 180,E1 -6931.675,E2 -6931.675} C_VEL
LIN {X 0,Y 480.891,Z 555.81,A -85,B 0,C 180,E1 -6933.351,E2 -6933.351} C_VEL
LIN {X 0,Y 480.854,Z 552.895,A -85,B 0,C 180,E1 -6934.611,E2 -6934.611} C_VEL
LIN {X 0,Y 481.022,Z 548.948,A -85,B 0,C 180,E1 -6935.87,E2 -6935.87} C_VEL
LIN {X 0,Y 481.116,Z 542.876,A -85,B 0,C 180,E1 -6937.343,E2 -6937.343} C_VEL
LIN {X 0,Y 481.426,Z 536.236,A -85,B 0,C 180,E1 -6938.606,E2 -6938.606} C_VEL
LIN {X 0,Y 481.753,Z 527.992,A -85,B 0,C 180,E1 -6939.87,E2 -6939.87} C_VEL
LIN {X 0,Y 482.086,Z 519.54,A -85,B 0,C 180,E1 -6940.925,E2 -6940.925} C_VEL
LIN {X 0,Y 482.601,Z 509.092,A -85,B 0,C 180,E1 -6941.977,E2 -6941.977} C_VEL
LIN {X 0,Y 483.005,Z 497.366,A -85,B 0,C 180,E1 -6942.924,E2 -6942.924} C_VEL
LIN {X 0,Y 483.473,Z 485.486,A -85,B 0,C 180,E1 -6943.663,E2 -6943.663} C_VEL
LIN {X 0,Y 483.865,Z 473.164,A -85,B 0,C 180,E1 -6944.242,E2 -6944.242} C_VEL
LIN {X 0,Y 483.824,Z 466.303,A -85,B 0,C 180,E1 -6944.498,E2 -6944.498} C_VEL
LIN {X 0,Y 481.644,Z 453.334,A -85,B 0,C 180,E1 -6944.908,E2 -6944.908} C_VEL
LIN {X 0,Y 481.337,Z 451.53,A -85,B 0,C 180,E1 -6944.967,E2 -6944.967} C_VEL
LIN {X 0,Y 481.556,Z 442.71,A -85,B 0,C 180,E1 -6947.847,E2 -6947.847} C_VEL
LIN {X 0,Y 481.797,Z 432.926,A -85,B 0,C 180,E1 -6951.001,E2 -6951.001} C_VEL
LIN {X 0,Y 482.029,Z 423.535,A -85,B 0,C 180,E1 -6954.094,E2 -6954.094} C_VEL
LIN {X 0,Y 482.433,Z 414.09,A -85,B 0,C 180,E1 -6957.297,E2 -6957.297} C_VEL
LIN {X 0,Y 482.755,Z 404.074,A -85,B 0,C 180,E1 -6960.803,E2 -6960.803} C_VEL
LIN {X 0,Y 483.133,Z 395.277,A -85,B 0,C 180,E1 -6963.987,E2 -6963.987} C_VEL
LIN {X 0,Y 483.25,Z 389.724,A -85,B 0,C 180,E1 -6966.086,E2 -6966.086} C_VEL
LIN {X 0,Y 482.162,Z 383.115,A -85,B 0,C 180,E1 -6968.812,E2 -6968.812} C_VEL
LIN {X 0,Y 481.685,Z 380.488,A -85,B 0,C 180,E1 -6970.005,E2 -6970.005} C_VEL
LIN {X 0,Y 481.669,Z 380.491,A -85,B 0,C 180,E1 -6973.297,E2 -6973.297} C_VEL
LIN {X 0,Y 481.661,Z 380.494,A -85,B 0,C 180,E1 -6975.641,E2 -6975.641} C_VEL
LIN {X 0,Y 481.659,Z 380.49,A -85,B 0,C 180,E1 -6978.958,E2 -6978.958} C_VEL
LIN {X 0,Y 481.659,Z 380.487,A -85,B 0,C 180,E1 -6981.993,E2 -6981.993} C_VEL
LIN {X 0,Y 481.695,Z 380.485,A -85,B 0,C 180,E1 -6985.318,E2 -6985.318} C_VEL
LIN {X 0,Y 481.648,Z 380.488,A -85,B 0,C 180,E1 -6988.312,E2 -6988.312} C_VEL
LIN {X 0,Y 481.703,Z 380.481,A -85,B 0,C 180,E1 -6991.219,E2 -6991.219} C_VEL
LIN {X 0,Y 481.693,Z 380.483,A -85,B 0,C 180,E1 -6994.042,E2 -6994.042} C_VEL
LIN {X 0,Y 481.677,Z 380.485,A -85,B 0,C 180,E1 -6996.812,E2 -6996.812} C_VEL
LIN {X 0,Y 481.701,Z 380.482,A -85,B 0,C 180,E1 -6999.503,E2 -6999.503} C_VEL
LIN {X 0,Y 481.711,Z 380.48,A -85,B 0,C 180,E1 -7002.159,E2 -7002.159} C_VEL
LIN {X 0,Y 481.747,Z 380.477,A -85,B 0,C 180,E1 -7004.776,E2 -7004.776} C_VEL
LIN {X 0,Y 481.799,Z 380.473,A -85,B 0,C 180,E1 -7008.216,E2 -7008.216} C_VEL
LIN {X 0,Y 481.767,Z 380.474,A -85,B 0,C 180,E1 -7011.612,E2 -7011.612} C_VEL
LIN {X 0,Y 481.82,Z 380.467,A -85,B 0,C 180,E1 -7014.14,E2 -7014.14} C_VEL
LIN {X 0,Y 481.931,Z 380.45,A -85,B 0,C 180,E1 -7017.493,E2 -7017.493} C_VEL
LIN {X 0,Y 481.909,Z 380.456,A -85,B 0,C 180,E1 -7020.836,E2 -7020.836} C_VEL
LIN {X 0,Y 481.93,Z 380.454,A -85,B 0,C 180,E1 -7022.507,E2 -7022.507} C_VEL
LIN {X 0,Y 481.82,Z 380.467,A -85,B 0,C 180,E1 -7025.86,E2 -7025.86} C_VEL
LIN {X 0,Y 481.765,Z 380.478,A -85,B 0,C 180,E1 -7028.388,E2 -7028.388} C_VEL
LIN {X 0,Y 481.755,Z 380.476,A -85,B 0,C 180,E1 -7031.785,E2 -7031.785} C_VEL
LIN {X 0,Y 481.747,Z 380.477,A -85,B 0,C 180,E1 -7035.224,E2 -7035.224} C_VEL
LIN {X 0,Y 481.713,Z 380.482,A -85,B 0,C 180,E1 -7038.722,E2 -7038.722} C_VEL
LIN {X 0,Y 481.649,Z 380.487,A -85,B 0,C 180,E1 -7041.395,E2 -7041.395} C_VEL
LIN {X 0,Y 481.665,Z 380.488,A -85,B 0,C 180,E1 -7044.114,E2 -7044.114} C_VEL
LIN {X 0,Y 481.751,Z 380.476,A -85,B 0,C 180,E1 -7047.139,E2 -7047.139} C_VEL
LIN {X 0,Y 481.682,Z 380.485,A -85,B 0,C 180,E1 -7049.741,E2 -7049.741} C_VEL
LIN {X 0,Y 481.675,Z 380.485,A -85,B 0,C 180,E1 -7052.674,E2 -7052.674} C_VEL
LIN {X 0,Y 481.64,Z 380.492,A -85,B 0,C 180,E1 -7055.709,E2 -7055.709} C_VEL
LIN {X 0,Y 481.675,Z 380.484,A -85,B 0,C 180,E1 -7058.859,E2 -7058.859} C_VEL
LIN {X 0,Y 481.656,Z 380.488,A -85,B 0,C 180,E1 -7061.913,E2 -7061.913} C_VEL
LIN {X 0,Y 481.657,Z 380.488,A -85,B 0,C 180,E1 -7064.458,E2 -7064.458} C_VEL
LIN {X 0,Y 481.692,Z 380.482,A -85,B 0,C 180,E1 -7066.846,E2 -7066.846} C_VEL
LIN {X 0,Y 481.68,Z 380.484,A -85,B 0,C 180,E1 -7070.06,E2 -7070.06} C_VEL
LIN {X 0,Y 481.616,Z 380.496,A -85,B 0,C 180,E1 -7073.252,E2 -7073.252} C_VEL
LIN {X 0,Y 481.514,Z 380.509,A -85,B 0,C 180,E1 -7075.303,E2 -7075.303} C_VEL
LIN {X 0,Y 481.281,Z 380.79,A -85,B 0,C 180,E1 -7077.883,E2 -7077.883} C_VEL
LIN {X 0,Y 481.22,Z 384.057,A -85,B 0,C 180,E1 -7081.196,E2 -7081.196} C_VEL
LIN {X 0,Y 481.123,Z 387.118,A -85,B 0,C 180,E1 -7084.262,E2 -7084.262} C_VEL
LIN {X 0,Y 481.079,Z 389.867,A -85,B 0,C 180,E1 -7086.979,E2 -7086.979} C_VEL
LIN {X 0,Y 481.019,Z 390.778,A -85,B 0,C 180,E1 -7087.873,E2 -7087.873} C_VEL
LIN {X 0,Y 480.321,Z 391.564,A -85,B 0,C 180,E1 -7088.565,E2 -7088.565} C_VEL
LIN {X 0,Y 477.437,Z 393.036,A -85,B 0,C 180,E1 -7089.686,E2 -7089.686} C_VEL
LIN {X 0,Y 475.026,Z 394.245,A -85,B 0,C 180,E1 -7090.59,E2 -7090.59} C_VEL
LIN {X 0,Y 474.01,Z 395.108,A -85,B 0,C 180,E1 -7091.289,E2 -7091.289} C_VEL
LIN {X 0,Y 473.937,Z 395.377,A -85,B 0,C 180,E1 -7091.526,E2 -7091.526} C_VEL
LIN {X 0,Y 473.929,Z 399.322,A -85,B 0,C 180,E1 -7094.917,E2 -7094.917} C_VEL
LIN {X 0,Y 477.052,Z 413.152,A -85,B 0,C 180,E1 -7095.443,E2 -7095.443} C_VEL
LIN {X 0,Y 476.976,Z 425.486,A -85,B 0,C 180,E1 -7095.984,E2 -7095.984} C_VEL
LIN {X 0,Y 476.553,Z 437.325,A -85,B 0,C 180,E1 -7096.678,E2 -7096.678} C_VEL
LIN {X 0,Y 476.111,Z 448.65,A -85,B 0,C 180,E1 -7097.533,E2 -7097.533} C_VEL
LIN {X 0,Y 475.672,Z 458.854,A -85,B 0,C 180,E1 -7098.495,E2 -7098.495} C_VEL
LIN {X 0,Y 475.209,Z 468.007,A -85,B 0,C 180,E1 -7099.562,E2 -7099.562} C_VEL
LIN {X 0,Y 474.811,Z 476.881,A -85,B 0,C 180,E1 -7100.844,E2 -7100.844} C_VEL
LIN {X 0,Y 474.447,Z 484.024,A -85,B 0,C 180,E1 -7102.125,E2 -7102.125} C_VEL
LIN {X 0,Y 474.209,Z 490.092,A -85,B 0,C 180,E1 -7103.502,E2 -7103.502} C_VEL
LIN {X 0,Y 473.894,Z 494.831,A -85,B 0,C 180,E1 -7104.895,E2 -7104.895} C_VEL
LIN {X 0,Y 473.992,Z 497.092,A -85,B 0,C 180,E1 -7105.748,E2 -7105.748} C_VEL
LIN {X 0,Y 473.912,Z 498.943,A -85,B 0,C 180,E1 -7106.599,E2 -7106.599} C_VEL
LIN {X 0,Y 473.881,Z 500.337,A -85,B 0,C 180,E1 -7107.45,E2 -7107.45} C_VEL
LIN {X 0,Y 473.692,Z 501.947,A -85,B 0,C 180,E1 -7109.15,E2 -7109.15} C_VEL
LIN {X 0,Y 473.676,Z 502.182,A -85,B 0,C 180,E1 -7110,E2 -7110} C_VEL
LIN {X 0,Y 473.761,Z 501.415,A -85,B 0,C 180,E1 -7111.7,E2 -7111.7} C_VEL
LIN {X 0,Y 473.881,Z 500.451,A -85,B 0,C 180,E1 -7112.55,E2 -7112.55} C_VEL
LIN {X 0,Y 473.913,Z 499.107,A -85,B 0,C 180,E1 -7113.401,E2 -7113.401} C_VEL
LIN {X 0,Y 473.964,Z 496.266,A -85,B 0,C 180,E1 -7114.678,E2 -7114.678} C_VEL
LIN {X 0,Y 474.104,Z 492.408,A -85,B 0,C 180,E1 -7115.956,E2 -7115.956} C_VEL
LIN {X 0,Y 474.255,Z 487.432,A -85,B 0,C 180,E1 -7117.236,E2 -7117.236} C_VEL
LIN {X 0,Y 474.574,Z 481.159,A -85,B 0,C 180,E1 -7118.516,E2 -7118.516} C_VEL
LIN {X 0,Y 474.905,Z 473.305,A -85,B 0,C 180,E1 -7119.799,E2 -7119.799} C_VEL
LIN {X 0,Y 475.427,Z 463.522,A -85,B 0,C 180,E1 -7121.08,E2 -7121.08} C_VEL
LIN {X 0,Y 475.933,Z 453.252,A -85,B 0,C 180,E1 -7122.148,E2 -7122.148} C_VEL
LIN {X 0,Y 476.354,Z 441.746,A -85,B 0,C 180,E1 -7123.105,E2 -7123.105} C_VEL
LIN {X 0,Y 476.792,Z 430.119,A -85,B 0,C 180,E1 -7123.859,E2 -7123.859} C_VEL
LIN {X 0,Y 477.145,Z 418.104,A -85,B 0,C 180,E1 -7124.447,E2 -7124.447} C_VEL
LIN {X 0,Y 477.02,Z 412.742,A -85,B 0,C 180,E1 -7124.664,E2 -7124.664} C_VEL
LIN {X 0,Y 473.933,Z 399.253,A -85,B 0,C 180,E1 -7125.188,E2 -7125.188} C_VEL
LIN {X 0,Y 473.92,Z 395.615,A -85,B 0,C 180,E1 -7128.361,E2 -7128.361} C_VEL
LIN {X 0,Y 473.937,Z 392.849,A -85,B 0,C 180,E1 -7130.896,E2 -7130.896} C_VEL
LIN {X 0,Y 474.012,Z 390.048,A -85,B 0,C 180,E1 -7133.598,E2 -7133.598} C_VEL
LIN {X 0,Y 474.062,Z 387.194,A -85,B 0,C 180,E1 -7136.408,E2 -7136.408} C_VEL
LIN {X 0,Y 474.148,Z 384.389,A -85,B 0,C 180,E1 -7139.284,E2 -7139.284} C_VEL
LIN {X 0,Y 474.229,Z 381.415,A -85,B 0,C 180,E1 -7142.356,E2 -7142.356} C_VEL
LIN {X 0,Y 474.538,Z 381.374,A -85,B 0,C 180,E1 -7145.456,E2 -7145.456} C_VEL
LIN {X 0,Y 474.614,Z 381.366,A -85,B 0,C 180,E1 -7148.458,E2 -7148.458} C_VEL
LIN {X 0,Y 474.632,Z 381.361,A -85,B 0,C 180,E1 -7150.959,E2 -7150.959} C_VEL
LIN {X 0,Y 474.61,Z 381.368,A -85,B 0,C 180,E1 -7154.105,E2 -7154.105} C_VEL
LIN {X 0,Y 474.61,Z 381.366,A -85,B 0,C 180,E1 -7157.065,E2 -7157.065} C_VEL
LIN {X 0,Y 474.632,Z 381.364,A -85,B 0,C 180,E1 -7160.352,E2 -7160.352} C_VEL
LIN {X 0,Y 474.597,Z 381.365,A -85,B 0,C 180,E1 -7163.677,E2 -7163.677} C_VEL
LIN {X 0,Y 474.647,Z 381.36,A -85,B 0,C 180,E1 -7166.78,E2 -7166.78} C_VEL
LIN {X 0,Y 474.61,Z 381.367,A -85,B 0,C 180,E1 -7169.77,E2 -7169.77} C_VEL
LIN {X 0,Y 474.702,Z 381.355,A -85,B 0,C 180,E1 -7172.68,E2 -7172.68} C_VEL
LIN {X 0,Y 474.646,Z 381.359,A -85,B 0,C 180,E1 -7175.506,E2 -7175.506} C_VEL
LIN {X 0,Y 474.676,Z 381.356,A -85,B 0,C 180,E1 -7179.186,E2 -7179.186} C_VEL
LIN {X 0,Y 474.651,Z 381.361,A -85,B 0,C 180,E1 -7181.884,E2 -7181.884} C_VEL
LIN {X 0,Y 474.705,Z 381.355,A -85,B 0,C 180,E1 -7184.544,E2 -7184.544} C_VEL
LIN {X 0,Y 474.71,Z 381.357,A -85,B 0,C 180,E1 -7188.038,E2 -7188.038} C_VEL
LIN {X 0,Y 474.717,Z 381.353,A -85,B 0,C 180,E1 -7191.486,E2 -7191.486} C_VEL
LIN {X 0,Y 474.783,Z 381.344,A -85,B 0,C 180,E1 -7194.052,E2 -7194.052} C_VEL
LIN {X 0,Y 474.897,Z 381.33,A -85,B 0,C 180,E1 -7197.455,E2 -7197.455} C_VEL
LIN {X 0,Y 474.917,Z 381.33,A -85,B 0,C 180,E1 -7200,E2 -7200} C_VEL
LIN {X 0,Y 474.899,Z 381.326,A -85,B 0,C 180,E1 -7202.545,E2 -7202.545} C_VEL
LIN {X 0,Y 474.784,Z 381.343,A -85,B 0,C 180,E1 -7205.948,E2 -7205.948} C_VEL
LIN {X 0,Y 474.734,Z 381.35,A -85,B 0,C 180,E1 -7208.513,E2 -7208.513} C_VEL
LIN {X 0,Y 474.745,Z 381.351,A -85,B 0,C 180,E1 -7211.961,E2 -7211.961} C_VEL
LIN {X 0,Y 474.685,Z 381.356,A -85,B 0,C 180,E1 -7215.768,E2 -7215.768} C_VEL
LIN {X 0,Y 474.669,Z 381.36,A -85,B 0,C 180,E1 -7219.01,E2 -7219.01} C_VEL
LIN {X 0,Y 474.593,Z 381.368,A -85,B 0,C 180,E1 -7221.729,E2 -7221.729} C_VEL
LIN {X 0,Y 474.645,Z 381.361,A -85,B 0,C 180,E1 -7224.494,E2 -7224.494} C_VEL
LIN {X 0,Y 474.704,Z 381.357,A -85,B 0,C 180,E1 -7227.338,E2 -7227.338} C_VEL
LIN {X 0,Y 474.609,Z 381.367,A -85,B 0,C 180,E1 -7230.81,E2 -7230.81} C_VEL
LIN {X 0,Y 474.641,Z 381.362,A -85,B 0,C 180,E1 -7233.984,E2 -7233.984} C_VEL
LIN {X 0,Y 474.576,Z 381.37,A -85,B 0,C 180,E1 -7236.899,E2 -7236.899} C_VEL
LIN {X 0,Y 474.632,Z 381.363,A -85,B 0,C 180,E1 -7239.647,E2 -7239.647} C_VEL
LIN {X 0,Y 474.619,Z 381.368,A -85,B 0,C 180,E1 -7242.934,E2 -7242.934} C_VEL
LIN {X 0,Y 474.619,Z 381.365,A -85,B 0,C 180,E1 -7245.896,E2 -7245.896} C_VEL
LIN {X 0,Y 474.636,Z 381.364,A -85,B 0,C 180,E1 -7249.04,E2 -7249.04} C_VEL
LIN {X 0,Y 474.679,Z 381.491,A -85,B 0,C 180,E1 -7249.808,E2 -7249.808} C_VEL
LIN {X 0,Y 475.925,Z 388.611,A -85,B 0,C 180,E1 -7252.885,E2 -7252.885} C_VEL
LIN {X 0,Y 476.304,Z 391.982,A -85,B 0,C 180,E1 -7254.247,E2 -7254.247} C_VEL
LIN {X 0,Y 476.051,Z 398.949,A -85,B 0,C 180,E1 -7256.891,E2 -7256.891} C_VEL
LIN {X 0,Y 475.649,Z 407.063,A -85,B 0,C 180,E1 -7259.843,E2 -7259.843} C_VEL
LIN {X 0,Y 475.392,Z 415.195,A -85,B 0,C 180,E1 -7262.723,E2 -7262.723} C_VEL
LIN {X 0,Y 474.986,Z 424.687,A -85,B 0,C 180,E1 -7265.99,E2 -7265.99} C_VEL
LIN {X 0,Y 474.713,Z 434.218,A -85,B 0,C 180,E1 -7269.187,E2 -7269.187} C_VEL
LIN {X 0,Y 474.47,Z 443.784,A -85,B 0,C 180,E1 -7272.323,E2 -7272.323} C_VEL
LIN {X 0,Y 474.311,Z 451.589,A -85,B 0,C 180,E1 -7274.827,E2 -7274.827} C_VEL
LIN {X 0,Y 476.609,Z 464.898,A -85,B 0,C 180,E1 -7275.231,E2 -7275.231} C_VEL
LIN {X 0,Y 477.079,Z 470.497,A -85,B 0,C 180,E1 -7275.442,E2 -7275.442} C_VEL
LIN {X 0,Y 476.697,Z 482.506,A -85,B 0,C 180,E1 -7275.975,E2 -7275.975} C_VEL
LIN {X 0,Y 476.211,Z 494.674,A -85,B 0,C 180,E1 -7276.7,E2 -7276.7} C_VEL
LIN {X 0,Y 475.811,Z 505.482,A -85,B 0,C 180,E1 -7277.524,E2 -7277.524} C_VEL
LIN {X 0,Y 475.363,Z 515.644,A -85,B 0,C 180,E1 -7278.487,E2 -7278.487} C_VEL
LIN {X 0,Y 474.881,Z 524.784,A -85,B 0,C 180,E1 -7279.555,E2 -7279.555} C_VEL
LIN {X 0,Y 474.482,Z 533.687,A -85,B 0,C 180,E1 -7280.838,E2 -7280.838} C_VEL
LIN {X 0,Y 474.153,Z 540.848,A -85,B 0,C 180,E1 -7282.119,E2 -7282.119} C_VEL
LIN {X 0,Y 473.977,Z 546.719,A -85,B 0,C 180,E1 -7283.444,E2 -7283.444} C_VEL
LIN {X 0,Y 473.846,Z 551.676,A -85,B 0,C 180,E1 -7284.894,E2 -7284.894} C_VEL
LIN {X 0,Y 473.752,Z 553.958,A -85,B 0,C 180,E1 -7285.746,E2 -7285.746} C_VEL
LIN {X 0,Y 473.799,Z 555.806,A -85,B 0,C 180,E1 -7286.598,E2 -7286.598} C_VEL
LIN {X 0,Y 473.695,Z 558.182,A -85,B 0,C 180,E1 -7288.3,E2 -7288.3} C_VEL
LIN {X 0,Y 473.688,Z 558.785,A -85,B 0,C 180,E1 -7289.15,E2 -7289.15} C_VEL
LIN {X 0,Y 473.669,Z 559,A -85,B 0,C 180,E1 -7290,E2 -7290} C_VEL
LIN {X 0,Y 473.688,Z 558.786,A -85,B 0,C 180,E1 -7290.85,E2 -7290.85} C_VEL
LIN {X 0,Y 473.724,Z 557.196,A -85,B 0,C 180,E1 -7292.551,E2 -7292.551} C_VEL
LIN {X 0,Y 473.799,Z 555.81,A -85,B 0,C 180,E1 -7293.401,E2 -7293.401} C_VEL
LIN {X 0,Y 473.775,Z 552.895,A -85,B 0,C 180,E1 -7294.68,E2 -7294.68} C_VEL
LIN {X 0,Y 473.941,Z 548.948,A -85,B 0,C 180,E1 -7295.958,E2 -7295.958} C_VEL
LIN {X 0,Y 474.049,Z 542.875,A -85,B 0,C 180,E1 -7297.454,E2 -7297.454} C_VEL
LIN {X 0,Y 474.377,Z 536.235,A -85,B 0,C 180,E1 -7298.734,E2 -7298.734} C_VEL
LIN {X 0,Y 474.749,Z 527.992,A -85,B 0,C 180,E1 -7300.017,E2 -7300.017} C_VEL
LIN {X 0,Y 475.103,Z 519.54,A -85,B 0,C 180,E1 -7301.087,E2 -7301.087} C_VEL
LIN {X 0,Y 475.657,Z 509.091,A -85,B 0,C 180,E1 -7302.155,E2 -7302.155} C_VEL
LIN {X 0,Y 476.043,Z 497.91,A -85,B 0,C 180,E1 -7303.075,E2 -7303.075} C_VEL
LIN {X 0,Y 476.506,Z 487.403,A -85,B 0,C 180,E1 -7303.758,E2 -7303.758} C_VEL
LIN {X 0,Y 476.916,Z 475.763,A -85,B 0,C 180,E1 -7304.345,E2 -7304.345} C_VEL
LIN {X 0,Y 476.903,Z 466.683,A -85,B 0,C 180,E1 -7304.699,E2 -7304.699} C_VEL
LIN {X 0,Y 474.634,Z 453.502,A -85,B 0,C 180,E1 -7305.128,E2 -7305.128} C_VEL
LIN {X 0,Y 474.284,Z 451.434,A -85,B 0,C 180,E1 -7305.194,E2 -7305.194} C_VEL
LIN {X 0,Y 474.55,Z 440.935,A -85,B 0,C 180,E1 -7308.589,E2 -7308.589} C_VEL
LIN {X 0,Y 474.801,Z 431.44,A -85,B 0,C 180,E1 -7311.719,E2 -7311.719} C_VEL
LIN {X 0,Y 475.091,Z 421.893,A -85,B 0,C 180,E1 -7314.936,E2 -7314.936} C_VEL
LIN {X 0,Y 475.421,Z 413.621,A -85,B 0,C 180,E1 -7317.822,E2 -7317.822} C_VEL
LIN {X 0,Y 475.779,Z 404.349,A -85,B 0,C 180,E1 -7321.132,E2 -7321.132} C_VEL
LIN {X 0,Y 476.184,Z 395.871,A -85,B 0,C 180,E1 -7324.258,E2 -7324.258} C_VEL
LIN {X 0,Y 476.258,Z 390.895,A -85,B 0,C 180,E1 -7326.176,E2 -7326.176} C_VEL
LIN {X 0,Y 475.159,Z 384.296,A -85,B 0,C 180,E1 -7328.947,E2 -7328.947} C_VEL
LIN {X 0,Y 474.667,Z 381.361,A -85,B 0,C 180,E1 -7330.259,E2 -7330.259} C_VEL
LIN {X 0,Y 474.625,Z 381.37,A -85,B 0,C 180,E1 -7333.484,E2 -7333.484} C_VEL
LIN {X 0,Y 474.604,Z 381.365,A -85,B 0,C 180,E1 -7336.519,E2 -7336.519} C_VEL
LIN {X 0,Y 474.62,Z 381.363,A -85,B 0,C 180,E1 -7339.342,E2 -7339.342} C_VEL
LIN {X 0,Y 474.613,Z 381.365,A -85,B 0,C 180,E1 -7341.704,E2 -7341.704} C_VEL
LIN {X 0,Y 474.632,Z 381.363,A -85,B 0,C 180,E1 -7344.726,E2 -7344.726} C_VEL
LIN {X 0,Y 474.639,Z 381.361,A -85,B 0,C 180,E1 -7347.788,E2 -7347.788} C_VEL
LIN {X 0,Y 474.628,Z 381.366,A -85,B 0,C 180,E1 -7350.884,E2 -7350.884} C_VEL
LIN {X 0,Y 474.657,Z 381.358,A -85,B 0,C 180,E1 -7353.628,E2 -7353.628} C_VEL
LIN {X 0,Y 474.638,Z 381.362,A -85,B 0,C 180,E1 -7356.642,E2 -7356.642} C_VEL
LIN {X 0,Y 474.661,Z 381.359,A -85,B 0,C 180,E1 -7360.09,E2 -7360.09} C_VEL
LIN {X 0,Y 474.655,Z 381.363,A -85,B 0,C 180,E1 -7362.775,E2 -7362.775} C_VEL
LIN {X 0,Y 474.652,Z 381.358,A -85,B 0,C 180,E1 -7365.421,E2 -7365.421} C_VEL
LIN {X 0,Y 474.743,Z 381.35,A -85,B 0,C 180,E1 -7368.039,E2 -7368.039} C_VEL
LIN {X 0,Y 474.732,Z 381.35,A -85,B 0,C 180,E1 -7371.487,E2 -7371.487} C_VEL
LIN {X 0,Y 474.782,Z 381.343,A -85,B 0,C 180,E1 -7374.052,E2 -7374.052} C_VEL
LIN {X 0,Y 474.897,Z 381.326,A -85,B 0,C 180,E1 -7377.455,E2 -7377.455} C_VEL
LIN {X 0,Y 474.916,Z 381.33,A -85,B 0,C 180,E1 -7380,E2 -7380} C_VEL
LIN {X 0,Y 474.896,Z 381.33,A -85,B 0,C 180,E1 -7382.545,E2 -7382.545} C_VEL
LIN {X 0,Y 474.783,Z 381.344,A -85,B 0,C 180,E1 -7385.948,E2 -7385.948} C_VEL
LIN {X 0,Y 474.73,Z 381.352,A -85,B 0,C 180,E1 -7388.514,E2 -7388.514} C_VEL
LIN {X 0,Y 474.709,Z 381.356,A -85,B 0,C 180,E1 -7391.962,E2 -7391.962} C_VEL
LIN {X 0,Y 474.704,Z 381.355,A -85,B 0,C 180,E1 -7395.456,E2 -7395.456} C_VEL
LIN {X 0,Y 474.667,Z 381.358,A -85,B 0,C 180,E1 -7399.01,E2 -7399.01} C_VEL
LIN {X 0,Y 474.592,Z 381.367,A -85,B 0,C 180,E1 -7401.729,E2 -7401.729} C_VEL
LIN {X 0,Y 474.645,Z 381.36,A -85,B 0,C 180,E1 -7404.494,E2 -7404.494} C_VEL
LIN {X 0,Y 474.703,Z 381.355,A -85,B 0,C 180,E1 -7407.339,E2 -7407.339} C_VEL
LIN {X 0,Y 474.608,Z 381.366,A -85,B 0,C 180,E1 -7410.81,E2 -7410.81} C_VEL
LIN {X 0,Y 474.641,Z 381.365,A -85,B 0,C 180,E1 -7413.984,E2 -7413.984} C_VEL
LIN {X 0,Y 474.575,Z 381.367,A -85,B 0,C 180,E1 -7416.899,E2 -7416.899} C_VEL
LIN {X 0,Y 474.631,Z 381.365,A -85,B 0,C 180,E1 -7419.648,E2 -7419.648} C_VEL
LIN {X 0,Y 474.609,Z 381.366,A -85,B 0,C 180,E1 -7422.935,E2 -7422.935} C_VEL
LIN {X 0,Y 474.618,Z 381.367,A -85,B 0,C 180,E1 -7425.896,E2 -7425.896} C_VEL
LIN {X 0,Y 474.635,Z 381.36,A -85,B 0,C 180,E1 -7429.04,E2 -7429.04} C_VEL
LIN {X 0,Y 474.61,Z 381.366,A -85,B 0,C 180,E1 -7431.704,E2 -7431.704} C_VEL
LIN {X 0,Y 474.537,Z 381.375,A -85,B 0,C 180,E1 -7434.718,E2 -7434.718} C_VEL
LIN {X 0,Y 474.225,Z 381.417,A -85,B 0,C 180,E1 -7437.756,E2 -7437.756} C_VEL
LIN {X 0,Y 474.148,Z 384.574,A -85,B 0,C 180,E1 -7440.989,E2 -7440.989} C_VEL
LIN {X 0,Y 474.064,Z 387.16,A -85,B 0,C 180,E1 -7443.593,E2 -7443.593} C_VEL
LIN {X 0,Y 474.017,Z 389.958,A -85,B 0,C 180,E1 -7446.402,E2 -7446.402} C_VEL
LIN {X 0,Y 473.953,Z 392.798,A -85,B 0,C 180,E1 -7449.152,E2 -7449.152} C_VEL
LIN {X 0,Y 473.937,Z 395.377,A -85,B 0,C 180,E1 -7451.526,E2 -7451.526} C_VEL
LIN {X 0,Y 473.264,Z 395.967,A -85,B 0,C 180,E1 -7451.993,E2 -7451.993} C_VEL
LIN {X 0,Y 470.385,Z 397.08,A -85,B 0,C 180,E1 -7452.719,E2 -7452.719} C_VEL
LIN {X 0,Y 467.493,Z 398.214,A -85,B 0,C 180,E1 -7453.454,E2 -7453.454} C_VEL
LIN {X 0,Y 466.821,Z 398.837,A -85,B 0,C 180,E1 -7453.93,E2 -7453.93} C_VEL
LIN {X 0,Y 466.895,Z 399.897,A -85,B 0,C 180,E1 -7454.698,E2 -7454.698} C_VEL
LIN {X 0,Y 470.061,Z 413.39,A -85,B 0,C 180,E1 -7455.214,E2 -7455.214} C_VEL
LIN {X 0,Y 470.324,Z 417.683,A -85,B 0,C 180,E1 -7455.395,E2 -7455.395} C_VEL
LIN {X 0,Y 469.992,Z 428.911,A -85,B 0,C 180,E1 -7455.937,E2 -7455.937} C_VEL
LIN {X 0,Y 469.615,Z 439.452,A -85,B 0,C 180,E1 -7456.596,E2 -7456.596} C_VEL
LIN {X 0,Y 469.15,Z 450.365,A -85,B 0,C 180,E1 -7457.455,E2 -7457.455} C_VEL
LIN {X 0,Y 468.746,Z 459.289,A -85,B 0,C 180,E1 -7458.322,E2 -7458.322} C_VEL
LIN {X 0,Y 468.231,Z 468.443,A -85,B 0,C 180,E1 -7459.405,E2 -7459.405} C_VEL
LIN {X 0,Y 467.821,Z 477.315,A -85,B 0,C 180,E1 -7460.706,E2 -7460.706} C_VEL
LIN {X 0,Y 467.411,Z 484.459,A -85,B 0,C 180,E1 -7462.005,E2 -7462.005} C_VEL
LIN {X 0,Y 467.168,Z 490.759,A -85,B 0,C 180,E1 -7463.467,E2 -7463.467} C_VEL
LIN {X 0,Y 466.832,Z 495.264,A -85,B 0,C 180,E1 -7464.818,E2 -7464.818} C_VEL
LIN {X 0,Y 466.936,Z 497.524,A -85,B 0,C 180,E1 -7465.684,E2 -7465.684} C_VEL
LIN {X 0,Y 466.844,Z 499.376,A -85,B 0,C 180,E1 -7466.548,E2 -7466.548} C_VEL
LIN {X 0,Y 466.824,Z 500.768,A -85,B 0,C 180,E1 -7467.411,E2 -7467.411} C_VEL
LIN {X 0,Y 466.623,Z 502.378,A -85,B 0,C 180,E1 -7469.137,E2 -7469.137} C_VEL
LIN {X 0,Y 466.605,Z 502.613,A -85,B 0,C 180,E1 -7470,E2 -7470} C_VEL
LIN {X 0,Y 466.699,Z 501.845,A -85,B 0,C 180,E1 -7471.726,E2 -7471.726} C_VEL
LIN {X 0,Y 466.824,Z 500.88,A -85,B 0,C 180,E1 -7472.589,E2 -7472.589} C_VEL
LIN {X 0,Y 466.844,Z 499.537,A -85,B 0,C 180,E1 -7473.452,E2 -7473.452} C_VEL
LIN {X 0,Y 466.904,Z 496.696,A -85,B 0,C 180,E1 -7474.749,E2 -7474.749} C_VEL
LIN {X 0,Y 467.06,Z 492.838,A -85,B 0,C 180,E1 -7476.046,E2 -7476.046} C_VEL
LIN {X 0,Y 467.228,Z 487.861,A -85,B 0,C 180,E1 -7477.346,E2 -7477.346} C_VEL
LIN {X 0,Y 467.567,Z 481.588,A -85,B 0,C 180,E1 -7478.645,E2 -7478.645} C_VEL
LIN {X 0,Y 467.936,Z 473.732,A -85,B 0,C 180,E1 -7479.946,E2 -7479.946} C_VEL
LIN {X 0,Y 468.47,Z 463.95,A -85,B 0,C 180,E1 -7481.246,E2 -7481.246} C_VEL
LIN {X 0,Y 469.001,Z 453.679,A -85,B 0,C 180,E1 -7482.33,E2 -7482.33} C_VEL
LIN {X 0,Y 469.449,Z 443.282,A -85,B 0,C 180,E1 -7483.214,E2 -7483.214} C_VEL
LIN {X 0,Y 469.863,Z 432.36,A -85,B 0,C 180,E1 -7483.957,E2 -7483.957} C_VEL
LIN {X 0,Y 470.255,Z 419.82,A -85,B 0,C 180,E1 -7484.608,E2 -7484.608} C_VEL
LIN {X 0,Y 470.282,Z 414.499,A -85,B 0,C 180,E1 -7484.829,E2 -7484.829} C_VEL
LIN {X 0,Y 467.278,Z 401.589,A -85,B 0,C 180,E1 -7485.338,E2 -7485.338} C_VEL
LIN {X 0,Y 466.865,Z 399.655,A -85,B 0,C 180,E1 -7485.425,E2 -7485.425} C_VEL
LIN {X 0,Y 466.855,Z 396.158,A -85,B 0,C 180,E1 -7488.486,E2 -7488.486} C_VEL
LIN {X 0,Y 466.884,Z 393.242,A -85,B 0,C 180,E1 -7491.179,E2 -7491.179} C_VEL
LIN {X 0,Y 466.946,Z 390.369,A -85,B 0,C 180,E1 -7493.978,E2 -7493.978} C_VEL
LIN {X 0,Y 467.013,Z 387.482,A -85,B 0,C 180,E1 -7496.838,E2 -7496.838} C_VEL
LIN {X 0,Y 467.087,Z 384.647,A -85,B 0,C 180,E1 -7499.771,E2 -7499.771} C_VEL
LIN {X 0,Y 467.131,Z 382.703,A -85,B 0,C 180,E1 -7501.775,E2 -7501.775} C_VEL
LIN {X 0,Y 467.222,Z 382.288,A -85,B 0,C 180,E1 -7502.787,E2 -7502.787} C_VEL
LIN {X 0,Y 467.496,Z 382.251,A -85,B 0,C 180,E1 -7505.728,E2 -7505.728} C_VEL
LIN {X 0,Y 467.564,Z 382.246,A -85,B 0,C 180,E1 -7508.591,E2 -7508.591} C_VEL
LIN {X 0,Y 467.58,Z 382.238,A -85,B 0,C 180,E1 -7511.403,E2 -7511.403} C_VEL
LIN {X 0,Y 467.556,Z 382.244,A -85,B 0,C 180,E1 -7513.821,E2 -7513.821} C_VEL
LIN {X 0,Y 467.555,Z 382.245,A -85,B 0,C 180,E1 -7516.255,E2 -7516.255} C_VEL
LIN {X 0,Y 467.582,Z 382.244,A -85,B 0,C 180,E1 -7518.723,E2 -7518.723} C_VEL
LIN {X 0,Y 467.57,Z 382.242,A -85,B 0,C 180,E1 -7521.956,E2 -7521.956} C_VEL
LIN {X 0,Y 467.572,Z 382.24,A -85,B 0,C 180,E1 -7525.168,E2 -7525.168} C_VEL
LIN {X 0,Y 467.587,Z 382.241,A -85,B 0,C 180,E1 -7528.26,E2 -7528.26} C_VEL
LIN {X 0,Y 467.581,Z 382.241,A -85,B 0,C 180,E1 -7531.251,E2 -7531.251} C_VEL
LIN {X 0,Y 467.602,Z 382.241,A -85,B 0,C 180,E1 -7534.159,E2 -7534.159} C_VEL
LIN {X 0,Y 467.581,Z 382.238,A -85,B 0,C 180,E1 -7536.996,E2 -7536.996} C_VEL
LIN {X 0,Y 467.629,Z 382.238,A -85,B 0,C 180,E1 -7539.777,E2 -7539.777} C_VEL
LIN {X 0,Y 467.604,Z 382.24,A -85,B 0,C 180,E1 -7542.506,E2 -7542.506} C_VEL
LIN {X 0,Y 467.612,Z 382.238,A -85,B 0,C 180,E1 -7545.197,E2 -7545.197} C_VEL
LIN {X 0,Y 467.662,Z 382.233,A -85,B 0,C 180,E1 -7547.855,E2 -7547.855} C_VEL
LIN {X 0,Y 467.675,Z 382.229,A -85,B 0,C 180,E1 -7551.357,E2 -7551.357} C_VEL
LIN {X 0,Y 467.747,Z 382.22,A -85,B 0,C 180,E1 -7553.963,E2 -7553.963} C_VEL
LIN {X 0,Y 467.863,Z 382.206,A -85,B 0,C 180,E1 -7557.417,E2 -7557.417} C_VEL
LIN {X 0,Y 467.887,Z 382.205,A -85,B 0,C 180,E1 -7560,E2 -7560} C_VEL
LIN {X 0,Y 467.864,Z 382.203,A -85,B 0,C 180,E1 -7562.583,E2 -7562.583} C_VEL
LIN {X 0,Y 467.749,Z 382.22,A -85,B 0,C 180,E1 -7566.037,E2 -7566.037} C_VEL
LIN {X 0,Y 467.687,Z 382.228,A -85,B 0,C 180,E1 -7568.643,E2 -7568.643} C_VEL
LIN {X 0,Y 467.688,Z 382.228,A -85,B 0,C 180,E1 -7572.145,E2 -7572.145} C_VEL
LIN {X 0,Y 467.654,Z 382.231,A -85,B 0,C 180,E1 -7575.885,E2 -7575.885} C_VEL
LIN {X 0,Y 467.628,Z 382.237,A -85,B 0,C 180,E1 -7579.308,E2 -7579.308} C_VEL
LIN {X 0,Y 467.539,Z 382.247,A -85,B 0,C 180,E1 -7582.074,E2 -7582.074} C_VEL
LIN {X 0,Y 467.59,Z 382.24,A -85,B 0,C 180,E1 -7584.888,E2 -7584.888} C_VEL
LIN {X 0,Y 467.632,Z 382.234,A -85,B 0,C 180,E1 -7587.768,E2 -7587.768} C_VEL
LIN {X 0,Y 467.572,Z 382.246,A -85,B 0,C 180,E1 -7591.045,E2 -7591.045} C_VEL
LIN {X 0,Y 467.592,Z 382.24,A -85,B 0,C 180,E1 -7594.242,E2 -7594.242} C_VEL
LIN {X 0,Y 467.552,Z 382.246,A -85,B 0,C 180,E1 -7597.186,E2 -7597.186} C_VEL
LIN {X 0,Y 467.581,Z 382.239,A -85,B 0,C 180,E1 -7600.264,E2 -7600.264} C_VEL
LIN {X 0,Y 467.59,Z 382.244,A -85,B 0,C 180,E1 -7602.567,E2 -7602.567} C_VEL
LIN {X 0,Y 467.574,Z 382.243,A -85,B 0,C 180,E1 -7605.053,E2 -7605.053} C_VEL
LIN {X 0,Y 467.592,Z 382.242,A -85,B 0,C 180,E1 -7607.44,E2 -7607.44} C_VEL
LIN {X 0,Y 467.598,Z 382.252,A -85,B 0,C 180,E1 -7609.454,E2 -7609.454} C_VEL
LIN {X 0,Y 468.862,Z 389.388,A -85,B 0,C 180,E1 -7612.603,E2 -7612.603} C_VEL
LIN {X 0,Y 469.341,Z 393.415,A -85,B 0,C 180,E1 -7614.268,E2 -7614.268} C_VEL
LIN {X 0,Y 469.028,Z 400.647,A -85,B 0,C 180,E1 -7617.047,E2 -7617.047} C_VEL
LIN {X 0,Y 468.626,Z 408.204,A -85,B 0,C 180,E1 -7619.841,E2 -7619.841} C_VEL
LIN {X 0,Y 468.353,Z 416.331,A -85,B 0,C 180,E1 -7622.762,E2 -7622.762} C_VEL
LIN {X 0,Y 467.925,Z 425.785,A -85,B 0,C 180,E1 -7626.076,E2 -7626.076} C_VEL
LIN {X 0,Y 467.628,Z 435.264,A -85,B 0,C 180,E1 -7629.318,E2 -7629.318} C_VEL
LIN {X 0,Y 467.403,Z 443.471,A -85,B 0,C 180,E1 -7632.046,E2 -7632.046} C_VEL
LIN {X 0,Y 467.222,Z 451.058,A -85,B 0,C 180,E1 -7634.57,E2 -7634.57} C_VEL
LIN {X 0,Y 469.768,Z 466.329,A -85,B 0,C 180,E1 -7635.072,E2 -7635.072} C_VEL
LIN {X 0,Y 470.204,Z 470.184,A -85,B 0,C 180,E1 -7635.225,E2 -7635.225} C_VEL
LIN {X 0,Y 469.793,Z 482.242,A -85,B 0,C 180,E1 -7635.765,E2 -7635.765} C_VEL
LIN {X 0,Y 469.281,Z 494.472,A -85,B 0,C 180,E1 -7636.5,E2 -7636.5} C_VEL
LIN {X 0,Y 468.876,Z 504.97,A -85,B 0,C 180,E1 -7637.305,E2 -7637.305} C_VEL
